(* Logix 5000 project; controller test vendor 1 type 14 code 151 rev 32.13; software revision 32.02 *)

TASK P200ms_p10 (periodic, rate 200 ms, priority 10, watchdog 300 ms) : GUI, ValveProfile
TASK P_Sample_p5 (periodic, rate 10 ms, priority 5, watchdog 2000 ms) : measArray, ISR_ValveCtrl   // Get raw analog input and control of the breathing - MUST HAVE HIGHEST priority of all peridoc tasks
TASK P_Sample_p8 (periodic, rate 10 ms, priority 8, watchdog 500 ms) : Setup, calcBreath, initVent, BreathDetect, measCalc, MainFlow

MODULES
   Local : vendor 1 type 14 code 151 (Compact 0, rev 32.13)
      Counters : Embedded (Compact 3, rev 1.1, Output RPI 20 ms)
      Discrete_IO : Embedded (Compact 1, rev 3.1, Output RPI 20 ms)
      Analog_IO : Embedded (Compact 2, rev 1.1, Output RPI 2 ms)
END_MODULES

ADD_ON_INSTRUCTION AOI_ARRAYSHIFT   (* revision 1.0, vendor RA - Brian Askjaer *)
VAR_IN_OUT
   Inp_Array : REAL[1000,2]; {required}
   _Array : REAL[1000,2]; {required}
END_VAR

ROUTINE Logic   (* ladder *)
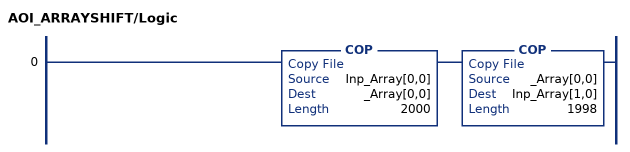
   0: COP(Inp_Array[0,0],_Array[0,0],2000)COP(_Array[0,0],Inp_Array[1,0],1998);
END_ROUTINE
END_ADD_ON_INSTRUCTION

ADD_ON_INSTRUCTION AOI_Ceil   (* revision 1.1 *)
VAR_INPUT
   In_X : REAL; {required}
END_VAR
VAR_IN_OUT
   Out_Ret : REAL; {required}
END_VAR
VAR
   _trunc : REAL; {access None}
   _aoiTrunc : AOI_Trunc; {access None}
   _n : DINT; {access None}
END_VAR

ROUTINE Logic   (* structured text *)
   AOI_Trunc( _aoiTrunc, In_X, _trunc );
   _n := _trunc;
   if _n < In_X then
   	_n := _n + 1;
   end_if;
   Out_Ret := _n;
   
END_ROUTINE
END_ADD_ON_INSTRUCTION

ADD_ON_INSTRUCTION AOI_FillArray_Real2D   (* revision 1.0, vendor RA - Brian Askjaer *)
VAR_IN_OUT
   Array : REAL[1000,2]; {required}
END_VAR
VAR_INPUT
   Source : DINT; {required}
   Len : DINT; {required}
END_VAR

ROUTINE Logic   (* ladder *)
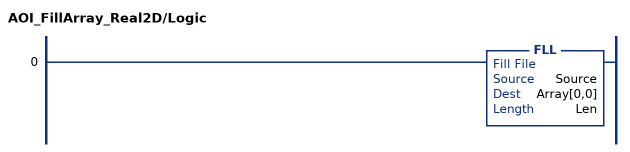
   0: FLL(Source,Array[0,0],Len);
END_ROUTINE
END_ADD_ON_INSTRUCTION

ADD_ON_INSTRUCTION AOI_FillArrayInt   (* revision 1.0, vendor RA - Brian Askjaer *)
VAR_IN_OUT
   Array : INT[1000]; {required}
END_VAR
VAR_INPUT
   Source : DINT; {required}
   Len : DINT; {required}
END_VAR

ROUTINE Logic   (* ladder *)
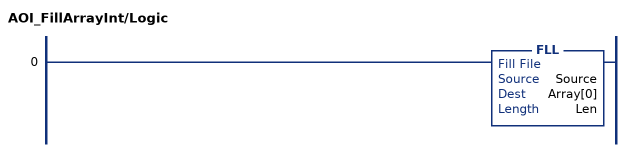
   0: FLL(Source,Array[0],Len);
END_ROUTINE
END_ADD_ON_INSTRUCTION

ADD_ON_INSTRUCTION AOI_FillArrayReal   (* revision 1.0, vendor RA - Brian Askjaer *)
VAR_IN_OUT
   Array : REAL[650]; {required}
END_VAR
VAR_INPUT
   Source : DINT; {required}
   Len : DINT; {required}
END_VAR

ROUTINE Logic   (* ladder *)
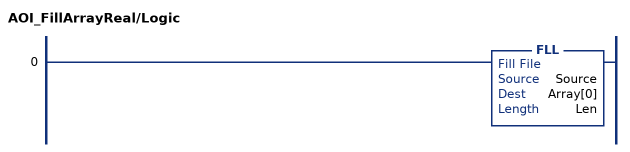
   0: FLL(Source,Array[0],Len);
END_ROUTINE
END_ADD_ON_INSTRUCTION

ADD_ON_INSTRUCTION AOI_FillArrayReal50   (* revision 1.0, vendor RA - Brian Askjaer *)
VAR_IN_OUT
   Array : REAL[50]; {required}
END_VAR
VAR_INPUT
   Source : DINT; {required}
   Len : DINT; {required}
END_VAR

ROUTINE Logic   (* ladder *)
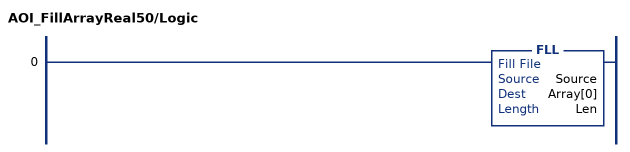
   0: FLL(Source,Array[0],Len);
END_ROUTINE
END_ADD_ON_INSTRUCTION

ADD_ON_INSTRUCTION AOI_FilterSignal   (* revision 1.1, ExecutePrescan *)
VAR_INPUT
   In_rRawSignal : REAL; {required}
   In_bInitialize : BOOL; {visible}
   Par_eType : DINT; {visible}   // 0: MEDIAN; 1: MEAN
   Par_nWindowLeft : DINT; {visible}
   Par_nWindowsRight : DINT; {visible}
   Par_bUseWeights : BOOL; {visible}   // Used for mean filtering
END_VAR
VAR_IN_OUT
   Par_rWeights : REAL[1]; {required}   // Used for mean filtering
END_VAR
VAR_OUTPUT
   Out_Buffering : BOOL; {visible}
   Out_rFilteredSignalDelayed : REAL; {access Read Only, visible}
   ER : BOOL; {access Read Only, visible}
   Err : DINT; {visible}
END_VAR
VAR
   _n1 : DINT; {access None}
   _n0 : DINT; {access None}
   _nN : DINT; {access None}
   _nM : DINT; {access None}
   _rWs : REAL[31]; {access None}
   _bW : BOOL; {access None}
   _idx : DINT; {access None}
   _bFirstScan : BOOL; {access None}
   _nTmp : DINT; {access None}
   _rRawBuf : REAL[31]; {access None}
   _eType : DINT; {access None}
   _srt : CONTROL; {access None}
   _nBufferUsage : DINT; {access None}
   _rBufSorted : REAL[31]; {access None}
   _i : DINT; {access None}
   _rSum : REAL; {access None}
   _w : REAL; {access None}
   _nOff : DINT; {access None}
   _n2 : DINT; {access None}
   _bOdd : BOOL; {access None}
   _rSumW : REAL; {access None}
END_VAR

ROUTINE Logic   (* structured text *)
   if ER and not ( _bFirstScan or In_bInitialize ) then
   	tnd();
   end_if;
   
   // Initialization
   if In_bInitialize or _bFirstScan then
   	ER  := 0;
   	Err := 0;
   	_idx := 0;
   	_nBufferUsage := 0;
   
   	// Validate parameters
   	_nTmp := Par_nWindowLeft + Par_nWindowsRight + 1;
   	if Par_nWindowLeft   < 0 then Err := 1; end_if;
   	if Par_nWindowsRight < 0 then Err := 2; end_if;
   	if _nTmp > _nM  then Err := 3; end_if;
   	if Par_eType <> 0 and Par_eType <> 1 then Err := 4; end_if;
   	if Err <> 0 then
   		ER := 1;
   		tnd();
   	end_if;
   
   	// Store parameters ( make filter behaviour independent from outside
   	//   parameters' changes ).
   	_bW := Par_bUseWeights;
   	_n0 := Par_nWindowLeft;
   	_n1 := Par_nWindowsRight;
   	_nN := _nTmp;
   	_n2 := _nN / 2;
   	_bOdd := ( _nN mod 2 ) = 1; // neighbourhood window composed of a odd number of points
   	_eType := Par_eType;
   	cop( Par_rWeights[0], _rWs[0], _nN );
   	_srt.POS := 0;
   	_srt.LEN := _nN;
   	_w := 1.0;
   	_rSumW := _nN;
   	if _bW then
   		_rSumW := 0.0;
   		for _i := 0 to _nN - 1 do
   			_rSumW := _rSumW + _rWs[_i];
   		end_for;
   	end_if;
   
   end_if;
   _bFirstScan := 0;
   In_bInitialize := 0;
   
   // While buffering data the filter isn't applied
   _rRawBuf[ _idx ] := In_rRawSignal;
   if _nBufferUsage < _nN then _nBufferUsage := _nBufferUsage + 1; end_if;
   Out_Buffering := _nBufferUsage <> _nN;
   
   if not Out_Buffering then
   
   	case _eType of
   
   		0: // MEDIAN
   		// Very simple implementation but not very efficient.
   		//   It's ok here because a single filtered value is
   		//   calculated at every scan of the plc.
   		// I'm using firmware instruction SRT to
   		//   sort the buffer array, because it's faster
   		//   than anything that could be implemented in
   		//   structure text. In case SRT isn't available in
   		//   other PLCs, a sorting algorithm could be implemented.
   		//   For example, in file sort/sort.c of the Gnu Scientific
   		//     Library (ftp://ftp.gnu.org/gnu/gsl/) there is an
   		//     implementation of the heap sort algorithm.
   		// TODO: replace the SRT instruction with such GLS
   		//       implementation so that this code can be reused
   		//       in any PLC.
   		cop( _rRawBuf[0], _rBufSorted[0], _nN );
   		SRT( _rBufSorted, 0, _srt );
   		if _bOdd then
   			Out_rFilteredSignalDelayed := _rBufSorted[_n2];
   		else
   			Out_rFilteredSignalDelayed := 0.5 * ( _rBufSorted[_n2-1] + _rBufSorted[_n2] );
   		end_if;
   
   		1: // MEAN
   		// Note: instruction MAVE could be used here, but I find
   		//       the following code clearer. Moreover the code
   		//       can be used in any PLC which doesn't include the
   		//       MAVE instruction.
   		_rSum := 0.0;
   		for _i := 0 to _nN - 1 do
   			if _bW then _w := _rWs[_i]; end_if;
   			_rSum := _rSum + _w * _rRawBuf[ ( _idx + 1 + _i ) mod _nN ];
   		end_for;
   		Out_rFilteredSignalDelayed := _rSum / _rSumW;
   
   	end_case;
   
   end_if;
   
   _idx := ( _idx + 1 ) mod _nN;
   
END_ROUTINE

ROUTINE Prescan   (* structured text *)
   // Calulate _nN = minimum between size( Par_rWeights ), size(_rWs), size(_rBuf) and size(_rBufSorted)
   size( _rWs, 0, _nM );
   size( _rRawBuf, 0, _nTmp );
   if _nTmp < _nM then _nM := _nTmp; end_if;
   size( _rBufSorted, 0, _nTmp );
   if _nTmp < _nM then _nM := _nTmp; end_if;
   size( Par_rWeights, 0, _nTmp );
   if _nTmp < _nM then _nM := _nTmp; end_if;
   
   // Used for initialization
   _bFirstScan := 1;
   
   // Data must be buffered at the beginning
   Out_Buffering := 1;
   
END_ROUTINE
END_ADD_ON_INSTRUCTION

ADD_ON_INSTRUCTION AOI_Floor   (* revision 1.1 *)
VAR_INPUT
   In_X : REAL; {required}
END_VAR
VAR_IN_OUT
   Out_Ret : REAL; {required}
END_VAR
VAR
   _n : DINT; {access None}
   _ret : REAL; {access None}
END_VAR

ROUTINE Logic   (* structured text *)
   _n := In_X;
   if In_X < _n then
   	_ret := _n - 1;
   else
   	_ret := _n;
   end_if;
   Out_Ret := _ret;
   
END_ROUTINE
END_ADD_ON_INSTRUCTION

ADD_ON_INSTRUCTION AOI_Max   (* revision 1.0, ExecutePrescan *)
VAR_IN_OUT
   In_Array : REAL[1000,2]; {required}
END_VAR
VAR_INPUT
   In_MainIndex : DINT; {required}
   In_N0 : INT; {required}
   In_N1 : INT; {required}
END_VAR
VAR_OUTPUT
   Out_Max : REAL; {visible}
   Err : DINT; {visible}
   ER : BOOL; {visible}
END_VAR
VAR_INPUT
   _i : DINT;
END_VAR
VAR
   _maxDim0 : DINT; {access None}
   _maxDim1 : DINT;
   _max : REAL; {access None}
   _tmp : REAL; {access None}
END_VAR

ROUTINE Logic   (* structured text *)
   ER  := 0;
   Err := 0;
   
   // Some checks
   if In_MainIndex < 0 or _maxDim1 <= In_MainIndex then Err := 1; end_if;
   if In_N0 < 0        or _maxDim0 <= In_N0        then Err := 2; end_if;
   if In_N1 < 0        or _maxDim0 <= In_N1        then Err := 3; end_if;
   if In_N0 > In_N1                                then Err := 4; end_if;
   if Err <> 0 then
   	ER := 1;
   	tnd();
   end_if;
   
   // Find maximum
   _max := In_Array[ In_N0, In_MainIndex ];
   for _i := In_N0 + 1 to In_N1 do
   	_tmp := In_Array[ _i, In_MainIndex ];
   	if _max < _tmp then _max := _tmp; end_if;
   end_for;
   Out_Max := _max;
   
END_ROUTINE

ROUTINE Prescan   (* structured text *)
   size( In_Array, 0, _maxDim0 ); // Dimension 0 is the most right index
   size( In_Array, 1, _maxDim1 );
   
END_ROUTINE
END_ADD_ON_INSTRUCTION

ADD_ON_INSTRUCTION AOI_Mean2D   (* revision 1.0, ExecutePrescan *)
VAR_IN_OUT
   In_Array : REAL[1000,2]; {required}
END_VAR
VAR_INPUT
   In_MainIndex : DINT; {required}
   In_N0 : INT; {required}
   In_N1 : INT; {required}
END_VAR
VAR_OUTPUT
   Out_Mean : REAL; {visible}
   Err : DINT; {visible}
   ER : BOOL; {visible}
END_VAR
VAR_INPUT
   _i : DINT;
END_VAR
VAR
   _maxDim0 : DINT; {access None}
   _maxDim1 : DINT;
   _sum : REAL; {access None}
END_VAR

ROUTINE Logic   (* structured text *)
   ER  := 0;
   Err := 0;
   
   // Some checks
   if In_MainIndex < 0 or _maxDim1 <= In_MainIndex then Err := 1; end_if;
   if In_N0 < 0        or _maxDim0 <= In_N0        then Err := 2; end_if;
   if In_N1 < 0        or _maxDim0 <= In_N1        then Err := 3; end_if;
   if In_N0 > In_N1                                then Err := 4; end_if;
   if Err <> 0 then
   	ER := 1;
   	tnd();
   end_if;
   
   // Find mean
   _sum := 0.0;
   for _i := In_N0 to In_N1 do
   	_sum := _sum + In_Array[ _i, In_MainIndex ];
   end_for;
   Out_Mean := _sum / ( In_N1 - In_N0 + 1 );
   
END_ROUTINE

ROUTINE Prescan   (* structured text *)
   size( In_Array, 0, _maxDim0 ); // Dimension 0 is the most right index
   size( In_Array, 1, _maxDim1 );
   
END_ROUTINE
END_ADD_ON_INSTRUCTION

ADD_ON_INSTRUCTION AOI_Mean50   (* revision 1.0, ExecutePrescan *)
VAR_IN_OUT
   In_Array : REAL[50]; {required}
END_VAR
VAR_INPUT
   In_N0 : INT; {required}
   In_N1 : INT; {required}
END_VAR
VAR_OUTPUT
   Out_Mean : REAL; {visible}
   Err : DINT; {visible}
   ER : BOOL; {visible}
END_VAR
VAR_INPUT
   _i : DINT;
END_VAR
VAR
   _maxDim0 : DINT; {access None}
   _maxDim1 : DINT;
   _sum : REAL; {access None}
END_VAR

ROUTINE Logic   (* structured text *)
   ER  := 0;
   Err := 0;
   
   // Some checks
   if In_N0 < 0        or _maxDim0 <= In_N0        then Err := 2; end_if;
   if In_N1 < 0        or _maxDim0 <= In_N1        then Err := 3; end_if;
   if In_N0 > In_N1                                then Err := 4; end_if;
   if Err <> 0 then
   	ER := 1;
   	tnd();
   end_if;
   
   // Find mean
   _sum := 0.0;
   for _i := In_N0 to In_N1 do
   	_sum := _sum + In_Array[ _i];
   end_for;
   Out_Mean := _sum / ( In_N1 - In_N0 + 1 );
   
END_ROUTINE

ROUTINE Prescan   (* structured text *)
   size( In_Array, 0, _maxDim0 ); // Dimension 0 is the most right index
   
END_ROUTINE
END_ADD_ON_INSTRUCTION

ADD_ON_INSTRUCTION AOI_Round   (* revision 1.0 *)
VAR_INPUT
   In_X : REAL; {required}
END_VAR
VAR_IN_OUT
   Out_Ret : REAL; {required}
END_VAR
VAR
   _n : DINT; {access None}
END_VAR

ROUTINE Logic   (* structured text *)
   _n := In_X;
   Out_Ret := _n;
   
END_ROUTINE
END_ADD_ON_INSTRUCTION

ADD_ON_INSTRUCTION AOI_Trunc   (* revision 1.0 *)
VAR_INPUT
   In_X : REAL; {required}
END_VAR
VAR_IN_OUT
   Out_Ret : REAL; {required}
END_VAR

ROUTINE Logic   (* structured text *)
   // TODO: Logix has a truc function but other PLCs may not.
   //       Replace the native function in Logix with an
   //       implementation which will work with other PLC.
   //       Note that AOI_Trunc and AOI_Ceil (which depends
   //       on AOI_Trunc ) may not be needed in the project.
   
   Out_Ret := trunc( In_X );
   
END_ROUTINE
END_ADD_ON_INSTRUCTION

VAR_GLOBAL   (* controller tags *)
   _CopDes1 : DINT;
   _CopDes4 : DINT;
   _CopDes5 : DINT;
   _CopDes6 : DINT;
   _CopDes8 : DINT;
   _CopLength : DINT;
   _CopLength1 : DINT;
   _CopLength3 : DINT;
   _CopLength4 : DINT;
   _CopLength5 : DINT;
   _CopLength6 : DINT;
   _CopLength7 : DINT := 2060;
   _CopLength8 : DINT;
   _CopSource : DINT;
   _CopSource1 : DINT;
   _CopSource3 : DINT;
   _CopSource4 : DINT;
   _CopSource5 : DINT;
   _CopSource6 : DINT;
   _CopSource7 : DINT := -30;
   _CopSource8 : DINT;
   _edbAoiFilterFlowAir : AOI_FilterSignal := (In_rRawSignal := 982.0, Par_nWindowLeft := 5, Par_nWindowsRight := 5, Out_rFilteredSignalDelayed := 982.0);
   _edbAoiFilterFlowO2 : AOI_FilterSignal := (In_rRawSignal := 983.0, Par_nWindowLeft := 5, Par_nWindowsRight := 5, Out_rFilteredSignalDelayed := 984.0);
   _edbAoiFilterPress : AOI_FilterSignal := (In_rRawSignal := 3963.0, Par_nWindowLeft := 5, Par_nWindowsRight := 5, Out_rFilteredSignalDelayed := 3951.0);
   _edbCanStore : BOOL := 1;
   _edbFlowArrFiltered : REAL[1000,2] := ([5,0] := 982.0, [6,0] := 982.0, [7,0] := 982.0, [8,0] := 982.0, [9,0] := 982.0, [10,0] := 982.0, [11,0] := 982.0, [12,0] := 982.0, [13,0] := 982.0, [14,0] := 982.0, [15,0] := 983.0, [16,0] := 983.0, [17,0] := 982.0, [18,0] := 982.0, [19,0] := 982.0, [20,0] := 982.0, [21,0] := 982.0, [22,0] := 982.0, [23,0] := 982.0, [24,0] := 982.0, [25,0] := 982.0, [26,0] := 982.0, [27,0] := 982.0, [28,0] := 982.0, [29,0] := 982.0, [30,0] := 982.0, [31,0] := 982.0, [32,0] := 982.0, [33,0] := 982.0, [34,0] := 982.0, [35,0] := 982.0, [36,0] := 982.0, [37,0] := 982.0, [38,0] := 982.0, [39,0] := 982.0, [40,0] := 982.0, [41,0] := 982.0, [42,0] := 982.0, [43,0] := 983.0, [44,0] := 983.0, [45,0] := 983.0, [46,0] := 983.0, [47,0] := 983.0, [48,0] := 983.0, [49,0] := 982.0, [50,0] := 982.0, [51,0] := 982.0, [52,0] := 982.0, [53,0] := 982.0, [54,0] := 982.0, [55,0] := 982.0, [56,0] := 982.0, [57,0] := 982.0, [58,0] := 982.0, [59,0] := 982.0, [60,0] := 982.0, [61,0] := 982.0, [62,0] := 982.0, [63,0] := 982.0, [64,0] := 982.0,
        [65,0] := 982.0, [66,0] := 982.0, [67,0] := 982.0, [68,0] := 982.0, [69,0] := 982.0, [70,0] := 982.0, [71,0] := 982.0, [72,0] := 982.0, [73,0] := 982.0, [74,0] := 982.0, [75,0] := 982.0, [76,0] := 982.0, [77,0] := 983.0, [78,0] := 983.0, [79,0] := 982.0, [80,0] := 982.0, [81,0] := 982.0, [82,0] := 982.0, [83,0] := 982.0, [84,0] := 982.0, [85,0] := 982.0, [86,0] := 982.0, [87,0] := 982.0, [88,0] := 982.0, [89,0] := 982.0, [90,0] := 982.0, [91,0] := 982.0, [92,0] := 982.0, [93,0] := 982.0, [94,0] := 982.0, [95,0] := 982.0, [96,0] := 982.0, [97,0] := 982.0, [98,0] := 982.0, [99,0] := 982.0, [100,0] := 982.0, [101,0] := 982.0, [102,0] := 982.0, [103,0] := 982.0, [104,0] := 982.0, [105,0] := 982.0, [106,0] := 982.0, [107,0] := 982.0, [108,0] := 982.0, [109,0] := 982.0, [110,0] := 982.0, [111,0] := 982.0, [112,0] := 982.0, [113,0] := 983.0, [114,0] := 983.0, [115,0] := 983.0, [116,0] := 983.0, [117,0] := 983.0, [118,0] := 982.0, [119,0] := 982.0, [120,0] := 982.0, [121,0] := 982.0, [122,0] := 982.0, [123,0] := 982.0, [124,0] := 982.0,
        [125,0] := 982.0, [126,0] := 982.0, [127,0] := 982.0, [128,0] := 982.0, [129,0] := 982.0, [130,0] := 982.0, [131,0] := 982.0, [132,0] := 982.0, [133,0] := 982.0, [134,0] := 982.0, [135,0] := 982.0, [136,0] := 982.0, [137,0] := 982.0, [138,0] := 982.0, [139,0] := 982.0, [140,0] := 982.0, [141,0] := 982.0, [142,0] := 982.0, [143,0] := 982.0, [144,0] := 983.0, [145,0] := 983.0, [146,0] := 983.0, [147,0] := 983.0, [148,0] := 983.0, [149,0] := 983.0, [150,0] := 982.0, [151,0] := 982.0, [152,0] := 982.0, [153,0] := 982.0, [154,0] := 982.0, [155,0] := 982.0, [156,0] := 982.0, [157,0] := 982.0, [158,0] := 982.0, [159,0] := 982.0, [160,0] := 982.0, [161,0] := 982.0, [162,0] := 982.0, [163,0] := 982.0, [164,0] := 982.0, [165,0] := 982.0, [166,0] := 982.0, [167,0] := 982.0, [168,0] := 982.0, [169,0] := 982.0, [170,0] := 982.0, [171,0] := 982.0, [172,0] := 982.0, [173,0] := 982.0, [174,0] := 982.0, [175,0] := 982.0, [176,0] := 983.0, [177,0] := 983.0, [178,0] := 983.0, [179,0] := 983.0, [180,0] := 982.0, [181,0] := 982.0, [182,0] := 982.0, [183,0] := 982.0, [184,0] := 982.0,
        [185,0] := 982.0, [186,0] := 982.0, [187,0] := 982.0, [188,0] := 982.0, [189,0] := 982.0, [190,0] := 982.0, [191,0] := 982.0, [192,0] := 982.0, [193,0] := 982.0, [194,0] := 982.0, [195,0] := 982.0, [196,0] := 982.0, [197,0] := 982.0, [198,0] := 982.0, [199,0] := 982.0, [200,0] := 982.0, [201,0] := 982.0, [202,0] := 982.0, [203,0] := 982.0, [204,0] := 982.0, [205,0] := 982.0, [206,0] := 982.0, [207,0] := 982.0, [208,0] := 982.0, [209,0] := 982.0, [210,0] := 982.0, [211,0] := 982.0, [212,0] := 982.0, [213,0] := 982.0, [214,0] := 982.0, [215,0] := 982.0, [216,0] := 982.0, [217,0] := 982.0, [218,0] := 982.0, [219,0] := 982.0, [220,0] := 982.0, [221,0] := 982.0, [222,0] := 982.0, [223,0] := 982.0, [224,0] := 982.0, [225,0] := 982.0, [226,0] := 982.0, [227,0] := 982.0, [228,0] := 982.0, [229,0] := 982.0, [230,0] := 982.0, [231,0] := 982.0, [232,0] := 982.0, [233,0] := 982.0, [234,0] := 982.0, [235,0] := 982.0, [236,0] := 982.0, [237,0] := 982.0, [238,0] := 982.0, [239,0] := 982.0, [240,0] := 982.0, [241,0] := 982.0, [242,0] := 982.0, [243,0] := 982.0, [244,0] := 982.0,
        [245,0] := 982.0, [246,0] := 982.0, [247,0] := 982.0, [248,0] := 982.0, [249,0] := 982.0, [250,0] := 982.0, [251,0] := 982.0, [252,0] := 982.0, [253,0] := 982.0, [254,0] := 982.0, [255,0] := 982.0, [256,0] := 982.0, [257,0] := 982.0, [258,0] := 982.0, [259,0] := 982.0, [260,0] := 982.0, [261,0] := 982.0, [262,0] := 982.0, [263,0] := 982.0, [264,0] := 982.0, [265,0] := 982.0, [266,0] := 982.0, [267,0] := 982.0, [268,0] := 982.0, [269,0] := 982.0, [270,0] := 982.0, [271,0] := 983.0, [272,0] := 983.0, [273,0] := 983.0, [274,0] := 983.0, [275,0] := 982.0, [276,0] := 982.0, [277,0] := 982.0, [278,0] := 982.0, [279,0] := 982.0, [280,0] := 982.0, [281,0] := 982.0, [282,0] := 982.0, [283,0] := 982.0, [284,0] := 982.0, [285,0] := 982.0, [286,0] := 982.0, [287,0] := 982.0, [288,0] := 982.0, [289,0] := 982.0, [290,0] := 982.0, [291,0] := 982.0, [292,0] := 982.0, [293,0] := 982.0, [294,0] := 982.0, [295,0] := 982.0, [296,0] := 982.0, [297,0] := 982.0, [298,0] := 982.0, [299,0] := 982.0, [300,0] := 982.0, [301,0] := 982.0, [302,0] := 982.0, [303,0] := 982.0, [304,0] := 982.0,
        [305,0] := 982.0, [306,0] := 982.0, [307,0] := 982.0, [308,0] := 982.0, [309,0] := 982.0, [310,0] := 982.0, [311,0] := 982.0, [312,0] := 982.0, [313,0] := 982.0, [314,0] := 982.0, [315,0] := 982.0, [316,0] := 982.0, [317,0] := 982.0, [318,0] := 982.0, [319,0] := 982.0, [320,0] := 982.0, [321,0] := 982.0, [322,0] := 982.0, [323,0] := 982.0, [324,0] := 982.0, [325,0] := 982.0, [326,0] := 982.0, [327,0] := 982.0, [328,0] := 982.0, [329,0] := 982.0, [330,0] := 982.0, [331,0] := 982.0, [332,0] := 983.0, [333,0] := 983.0, [334,0] := 983.0, [335,0] := 983.0, [336,0] := 983.0, [337,0] := 983.0, [338,0] := 983.0, [339,0] := 983.0, [340,0] := 982.0, [341,0] := 982.0, [342,0] := 982.0, [343,0] := 982.0, [344,0] := 982.0, [345,0] := 982.0, [346,0] := 982.0, [347,0] := 982.0, [348,0] := 982.0, [349,0] := 982.0, [350,0] := 982.0, [351,0] := 982.0, [352,0] := 982.0, [353,0] := 982.0, [354,0] := 982.0, [355,0] := 982.0, [356,0] := 982.0, [357,0] := 982.0, [358,0] := 982.0, [359,0] := 982.0, [360,0] := 982.0, [361,0] := 982.0, [362,0] := 982.0, [363,0] := 982.0, [364,0] := 982.0,
        [365,0] := 982.0, [366,0] := 982.0, [367,0] := 982.0, [368,0] := 982.0, [369,0] := 982.0, [370,0] := 982.0, [371,0] := 982.0, [372,0] := 982.0, [373,0] := 982.0, [374,0] := 982.0, [375,0] := 982.0, [376,0] := 982.0, [377,0] := 982.0, [378,0] := 982.0, [379,0] := 982.0, [380,0] := 982.0, [381,0] := 982.0, [382,0] := 982.0, [383,0] := 982.0, [384,0] := 982.0, [385,0] := 982.0, [386,0] := 982.0, [387,0] := 982.0, [388,0] := 982.0, [389,0] := 982.0, [390,0] := 982.0, [391,0] := 982.0, [392,0] := 982.0, [393,0] := 982.0, [394,0] := 982.0, [395,0] := 982.0, [396,0] := 982.0, [397,0] := 982.0, [398,0] := 982.0, [399,0] := 982.0, [400,0] := 982.0, [401,0] := 982.0, [402,0] := 982.0, [403,0] := 982.0, [404,0] := 982.0, [405,0] := 982.0, [406,0] := 982.0, [407,0] := 982.0, [408,0] := 982.0, [409,0] := 982.0, [410,0] := 982.0, [411,0] := 982.0, [412,0] := 982.0, [413,0] := 982.0, [414,0] := 982.0, [415,0] := 982.0, [416,0] := 982.0, [417,0] := 982.0, [418,0] := 982.0, [419,0] := 982.0, [420,0] := 982.0, [421,0] := 982.0, [422,0] := 982.0, [423,0] := 982.0, [424,0] := 982.0,
        [425,0] := 982.0, [426,0] := 983.0, [427,0] := 983.0, [428,0] := 983.0, [429,0] := 983.0, [430,0] := 983.0, [431,0] := 982.0, [432,0] := 982.0, [433,0] := 982.0, [434,0] := 982.0, [435,0] := 982.0, [436,0] := 982.0, [437,0] := 982.0, [438,0] := 982.0, [439,0] := 982.0, [440,0] := 982.0, [441,0] := 982.0, [442,0] := 982.0, [443,0] := 982.0, [444,0] := 982.0, [445,0] := 982.0, [446,0] := 982.0, [447,0] := 982.0, [448,0] := 982.0, [449,0] := 982.0, [450,0] := 982.0, [451,0] := 982.0, [452,0] := 982.0, [453,0] := 982.0, [454,0] := 982.0, [455,0] := 982.0, [456,0] := 982.0, [457,0] := 982.0, [458,0] := 982.0, [459,0] := 982.0, [460,0] := 982.0, [461,0] := 982.0, [462,0] := 982.0, [463,0] := 982.0, [464,0] := 982.0, [465,0] := 983.0, [466,0] := 983.0, [467,0] := 983.0, [468,0] := 983.0, [469,0] := 982.0, [470,0] := 982.0, [471,0] := 982.0, [472,0] := 982.0, [473,0] := 982.0, [474,0] := 982.0, [475,0] := 982.0, [476,0] := 982.0, [477,0] := 982.0, [478,0] := 982.0, [479,0] := 982.0, [480,0] := 982.0, [481,0] := 982.0, [482,0] := 982.0, [483,0] := 982.0, [484,0] := 982.0,
        [485,0] := 982.0, [486,0] := 982.0, [487,0] := 982.0, [488,0] := 982.0, [489,0] := 982.0, [490,0] := 982.0, [491,0] := 983.0, [492,0] := 983.0, [493,0] := 982.0, [494,0] := 982.0, [495,0] := 982.0, [496,0] := 982.0, [497,0] := 983.0, [498,0] := 983.0, [499,0] := 983.0, [500,0] := 982.0, [501,0] := 982.0, [502,0] := 982.0, [503,0] := 982.0, [504,0] := 982.0, [505,0] := 982.0, [506,0] := 982.0, [507,0] := 982.0, [508,0] := 982.0, [509,0] := 982.0, [510,0] := 982.0, [511,0] := 982.0, [512,0] := 982.0, [513,0] := 982.0, [514,0] := 982.0, [515,0] := 982.0, [516,0] := 982.0, [517,0] := 982.0, [518,0] := 982.0, [519,0] := 982.0, [520,0] := 982.0, [521,0] := 982.0, [522,0] := 982.0, [523,0] := 982.0, [524,0] := 982.0, [525,0] := 982.0, [526,0] := 982.0, [527,0] := 982.0, [528,0] := 982.0, [529,0] := 982.0, [530,0] := 983.0, [531,0] := 983.0, [532,0] := 982.0, [533,0] := 982.0, [534,0] := 982.0, [535,0] := 982.0, [536,0] := 982.0, [537,0] := 982.0, [538,0] := 982.0, [539,0] := 982.0, [540,0] := 982.0, [541,0] := 982.0, [542,0] := 982.0, [543,0] := 982.0, [544,0] := 982.0,
        [545,0] := 982.0, [546,0] := 982.0, [547,0] := 982.0, [548,0] := 982.0, [549,0] := 982.0, [550,0] := 982.0, [551,0] := 982.0, [552,0] := 982.0, [553,0] := 982.0, [554,0] := 982.0, [555,0] := 982.0, [556,0] := 982.0, [557,0] := 982.0, [558,0] := 982.0, [559,0] := 982.0, [560,0] := 982.0, [561,0] := 982.0, [562,0] := 982.0, [563,0] := 982.0, [564,0] := 982.0, [565,0] := 983.0, [566,0] := 983.0, [567,0] := 983.0, [568,0] := 983.0, [569,0] := 983.0, [570,0] := 983.0, [571,0] := 983.0, [572,0] := 983.0, [573,0] := 982.0, [574,0] := 982.0, [575,0] := 982.0, [576,0] := 982.0, [577,0] := 982.0, [578,0] := 982.0, [579,0] := 982.0, [580,0] := 982.0, [581,0] := 982.0, [582,0] := 982.0, [583,0] := 982.0, [584,0] := 982.0, [585,0] := 982.0, [586,0] := 982.0, [587,0] := 982.0, [588,0] := 982.0, [589,0] := 982.0, [590,0] := 982.0, [591,0] := 982.0, [592,0] := 982.0, [593,0] := 982.0, [594,0] := 982.0, [595,0] := 982.0, [596,0] := 982.0, [597,0] := 982.0, [598,0] := 982.0, [599,0] := 982.0, [600,0] := 982.0, [601,0] := 982.0, [602,0] := 982.0, [603,0] := 982.0, [604,0] := 982.0,
        [605,0] := 982.0, [606,0] := 982.0, [607,0] := 982.0, [608,0] := 982.0, [609,0] := 982.0, [610,0] := 982.0, [611,0] := 982.0, [612,0] := 982.0, [613,0] := 982.0, [614,0] := 982.0, [615,0] := 982.0, [616,0] := 982.0, [617,0] := 982.0, [618,0] := 982.0, [619,0] := 982.0, [620,0] := 982.0, [621,0] := 982.0, [622,0] := 982.0, [623,0] := 982.0, [624,0] := 982.0, [625,0] := 982.0, [626,0] := 982.0, [627,0] := 982.0, [628,0] := 982.0, [629,0] := 982.0, [630,0] := 982.0, [631,0] := 982.0, [632,0] := 982.0, [633,0] := 982.0, [634,0] := 982.0, [635,0] := 982.0, [636,0] := 982.0, [637,0] := 982.0, [638,0] := 982.0, [639,0] := 982.0, [640,0] := 982.0, [641,0] := 982.0, [642,0] := 982.0, [643,0] := 982.0, [644,0] := 982.0, [645,0] := 982.0, [646,0] := 982.0, [647,0] := 982.0, [648,0] := 982.0, [649,0] := 982.0, [650,0] := 982.0, [651,0] := 982.0, [652,0] := 982.0, [653,0] := 982.0, [654,0] := 982.0, [655,0] := 983.0, [656,0] := 983.0, [657,0] := 982.0, [658,0] := 982.0, [659,0] := 982.0, [660,0] := 982.0, [661,0] := 982.0, [662,0] := 982.0, [663,0] := 982.0, [664,0] := 982.0,
        [665,0] := 982.0, [666,0] := 982.0, [667,0] := 982.0, [668,0] := 982.0, [669,0] := 982.0, [670,0] := 982.0, [671,0] := 982.0, [672,0] := 982.0, [673,0] := 982.0, [674,0] := 982.0, [675,0] := 982.0, [676,0] := 982.0, [677,0] := 982.0, [678,0] := 982.0, [679,0] := 982.0, [680,0] := 982.0, [681,0] := 982.0, [682,0] := 982.0, [683,0] := 982.0, [684,0] := 982.0, [685,0] := 982.0, [686,0] := 982.0, [687,0] := 982.0, [688,0] := 982.0, [689,0] := 982.0, [690,0] := 982.0, [691,0] := 982.0, [692,0] := 983.0, [693,0] := 983.0, [694,0] := 983.0, [695,0] := 983.0, [696,0] := 983.0, [697,0] := 983.0, [698,0] := 982.0, [699,0] := 982.0, [700,0] := 982.0, [701,0] := 982.0, [702,0] := 982.0, [703,0] := 982.0, [704,0] := 982.0, [705,0] := 982.0, [706,0] := 982.0, [707,0] := 982.0, [708,0] := 982.0, [709,0] := 982.0, [710,0] := 982.0, [711,0] := 982.0, [712,0] := 982.0, [713,0] := 982.0, [714,0] := 982.0, [715,0] := 982.0, [716,0] := 982.0, [717,0] := 982.0, [718,0] := 982.0, [719,0] := 982.0, [720,0] := 982.0, [721,0] := 982.0, [722,0] := 983.0, [723,0] := 983.0, [724,0] := 983.0,
        [725,0] := 983.0, [726,0] := 983.0, [727,0] := 983.0, [728,0] := 982.0, [729,0] := 982.0, [730,0] := 982.0, [731,0] := 982.0, [732,0] := 982.0, [733,0] := 982.0, [734,0] := 982.0, [735,0] := 982.0, [736,0] := 982.0, [737,0] := 982.0, [738,0] := 982.0, [739,0] := 982.0, [740,0] := 982.0, [741,0] := 982.0, [742,0] := 982.0, [743,0] := 982.0, [744,0] := 982.0, [745,0] := 982.0, [746,0] := 982.0, [747,0] := 982.0, [748,0] := 982.0, [749,0] := 982.0, [750,0] := 982.0, [751,0] := 982.0, [752,0] := 982.0, [753,0] := 983.0, [754,0] := 983.0, [755,0] := 983.0, [756,0] := 983.0, [757,0] := 983.0, [758,0] := 983.0, [759,0] := 982.0, [760,0] := 982.0, [761,0] := 982.0, [762,0] := 982.0, [763,0] := 982.0, [764,0] := 982.0, [765,0] := 982.0, [766,0] := 982.0, [767,0] := 982.0, [768,0] := 982.0, [769,0] := 982.0, [770,0] := 982.0, [771,0] := 982.0, [772,0] := 982.0, [773,0] := 982.0, [774,0] := 982.0, [775,0] := 982.0, [776,0] := 982.0, [777,0] := 982.0, [778,0] := 982.0, [779,0] := 982.0, [780,0] := 982.0, [781,0] := 982.0, [782,0] := 982.0, [783,0] := 982.0, [784,0] := 982.0,
        [785,0] := 983.0, [786,0] := 983.0, [787,0] := 983.0, [788,0] := 983.0, [789,0] := 982.0, [790,0] := 982.0, [791,0] := 982.0, [792,0] := 982.0, [793,0] := 982.0, [794,0] := 982.0, [795,0] := 982.0, [796,0] := 982.0, [797,0] := 982.0, [798,0] := 982.0, [799,0] := 982.0, [800,0] := 982.0, [801,0] := 982.0, [802,0] := 982.0, [803,0] := 982.0, [804,0] := 982.0, [805,0] := 982.0, [806,0] := 982.0, [807,0] := 982.0, [808,0] := 982.0, [809,0] := 982.0, [810,0] := 982.0, [811,0] := 982.0, [812,0] := 982.0, [813,0] := 982.0, [814,0] := 982.0, [815,0] := 982.0, [816,0] := 983.0, [817,0] := 983.0, [818,0] := 983.0, [819,0] := 983.0, [820,0] := 983.0, [821,0] := 982.0, [822,0] := 982.0, [823,0] := 982.0, [824,0] := 982.0, [825,0] := 982.0, [826,0] := 982.0, [827,0] := 982.0, [828,0] := 982.0, [829,0] := 982.0, [830,0] := 982.0, [831,0] := 982.0, [832,0] := 982.0, [833,0] := 982.0, [834,0] := 982.0, [835,0] := 982.0, [836,0] := 982.0, [837,0] := 982.0, [838,0] := 982.0, [839,0] := 982.0, [840,0] := 982.0, [841,0] := 982.0, [842,0] := 982.0, [843,0] := 982.0, [844,0] := 982.0,
        [845,0] := 982.0, [846,0] := 982.0, [847,0] := 983.0, [848,0] := 983.0, [849,0] := 983.0, [850,0] := 983.0, [851,0] := 983.0, [852,0] := 983.0, [853,0] := 982.0, [854,0] := 982.0, [855,0] := 982.0, [856,0] := 982.0, [857,0] := 982.0, [858,0] := 982.0, [859,0] := 982.0, [860,0] := 982.0, [861,0] := 982.0, [862,0] := 982.0, [863,0] := 982.0, [864,0] := 982.0, [865,0] := 982.0, [866,0] := 982.0, [867,0] := 982.0, [868,0] := 982.0, [869,0] := 982.0, [870,0] := 982.0, [871,0] := 982.0, [872,0] := 982.0, [873,0] := 982.0, [874,0] := 982.0, [875,0] := 982.0, [876,0] := 982.0, [877,0] := 982.0, [878,0] := 982.0, [879,0] := 982.0, [880,0] := 982.0, [881,0] := 982.0, [882,0] := 982.0, [883,0] := 982.0, [884,0] := 982.0, [885,0] := 982.0, [886,0] := 982.0, [887,0] := 982.0, [888,0] := 982.0, [889,0] := 982.0, [890,0] := 982.0, [891,0] := 982.0, [892,0] := 982.0, [893,0] := 982.0, [894,0] := 982.0, [895,0] := 982.0, [896,0] := 982.0, [897,0] := 982.0, [898,0] := 982.0, [899,0] := 982.0, [900,0] := 982.0, [901,0] := 982.0, [902,0] := 982.0, [903,0] := 982.0, [904,0] := 982.0,
        [905,0] := 982.0, [906,0] := 983.0, [907,0] := 983.0, [908,0] := 982.0, [909,0] := 982.0, [910,0] := 982.0, [911,0] := 982.0, [912,0] := 982.0, [913,0] := 982.0, [914,0] := 982.0, [915,0] := 982.0, [916,0] := 982.0, [917,0] := 982.0, [918,0] := 982.0, [919,0] := 982.0, [920,0] := 982.0, [921,0] := 982.0, [922,0] := 982.0, [923,0] := 982.0, [924,0] := 982.0, [925,0] := 982.0, [926,0] := 982.0, [927,0] := 982.0, [928,0] := 982.0, [929,0] := 982.0, [930,0] := 982.0, [931,0] := 982.0, [932,0] := 982.0, [933,0] := 982.0, [934,0] := 982.0, [935,0] := 982.0, [936,0] := 982.0, [937,0] := 982.0, [938,0] := 982.0, [939,0] := 982.0, [940,0] := 982.0, [941,0] := 982.0, [942,0] := 982.0, [943,0] := 982.0, [944,0] := 982.0, [945,0] := 982.0, [946,0] := 982.0, [947,0] := 982.0, [948,0] := 982.0, [949,0] := 982.0, [950,0] := 982.0, [951,0] := 982.0, [952,0] := 982.0, [953,0] := 982.0, [954,0] := 982.0, [955,0] := 982.0, [956,0] := 982.0, [957,0] := 983.0, [958,0] := 983.0, [959,0] := 982.0, [960,0] := 982.0, [961,0] := 982.0, [962,0] := 982.0, [963,0] := 982.0, [964,0] := 982.0,
        [965,0] := 982.0, [966,0] := 982.0, [967,0] := 982.0, [968,0] := 982.0, [969,0] := 982.0, [970,0] := 982.0, [971,0] := 982.0, [972,0] := 982.0, [973,0] := 982.0, [974,0] := 982.0, [975,0] := 982.0, [976,0] := 982.0, [977,0] := 982.0, [978,0] := 982.0, [979,0] := 983.0, [980,0] := 983.0, [981,0] := 983.0, [982,0] := 983.0, [983,0] := 983.0, [984,0] := 983.0, [985,0] := 983.0, [986,0] := 983.0, [987,0] := 982.0, [988,0] := 982.0, [989,0] := 982.0, [990,0] := 982.0, [991,0] := 982.0, [992,0] := 982.0, [993,0] := 982.0);
   _edbFlowO2Filtered : REAL[1000,2] := ([5,0] := 3948.0, [6,0] := 3948.0, [7,0] := 3948.0, [8,0] := 3948.0, [9,0] := 3948.0, [10,0] := 3948.0, [11,0] := 3948.0, [12,0] := 3948.0, [13,0] := 3948.0, [14,0] := 3950.0, [15,0] := 3950.0, [16,0] := 3950.0, [17,0] := 3951.0, [18,0] := 3951.0, [19,0] := 3951.0, [20,0] := 3951.0, [21,0] := 3951.0, [22,0] := 3951.0, [23,0] := 3951.0, [24,0] := 3951.0, [25,0] := 3951.0, [26,0] := 3951.0, [27,0] := 3951.0, [28,0] := 3951.0, [29,0] := 3948.0, [30,0] := 3948.0, [31,0] := 3948.0, [32,0] := 3948.0, [33,0] := 3948.0, [34,0] := 3957.0, [35,0] := 3957.0, [36,0] := 3957.0, [37,0] := 3957.0, [38,0] := 3948.0, [39,0] := 3948.0, [40,0] := 3945.0, [41,0] := 3945.0, [42,0] := 3945.0, [43,0] := 3945.0, [44,0] := 3954.0, [45,0] := 3954.0, [46,0] := 3954.0, [47,0] := 3954.0, [48,0] := 3954.0, [49,0] := 3954.0, [50,0] := 3954.0, [51,0] := 3954.0, [52,0] := 3954.0, [53,0] := 3954.0, [54,0] := 3954.0, [55,0] := 3954.0, [56,0] := 3954.0, [57,0] := 3954.0, [58,0] := 3944.0, [59,0] := 3944.0, [60,0] := 3944.0, [61,0] := 3944.0, [62,0] := 3954.0, [63,0] := 3954.0, [64,0] := 3954.0,
        [65,0] := 3954.0, [66,0] := 3954.0, [67,0] := 3956.0, [68,0] := 3956.0, [69,0] := 3956.0, [70,0] := 3956.0, [71,0] := 3956.0, [72,0] := 3956.0, [73,0] := 3956.0, [74,0] := 3956.0, [75,0] := 3956.0, [76,0] := 3956.0, [77,0] := 3956.0, [78,0] := 3956.0, [79,0] := 3962.0, [80,0] := 3962.0, [81,0] := 3962.0, [82,0] := 3962.0, [83,0] := 3962.0, [84,0] := 3962.0, [85,0] := 3962.0, [86,0] := 3962.0, [87,0] := 3962.0, [88,0] := 3962.0, [89,0] := 3962.0, [90,0] := 3962.0, [91,0] := 3955.0, [92,0] := 3955.0, [93,0] := 3955.0, [94,0] := 3955.0, [95,0] := 3955.0, [96,0] := 3955.0, [97,0] := 3955.0, [98,0] := 3955.0, [99,0] := 3955.0, [100,0] := 3955.0, [101,0] := 3955.0, [102,0] := 3955.0, [103,0] := 3953.0, [104,0] := 3953.0, [105,0] := 3953.0, [106,0] := 3953.0, [107,0] := 3953.0, [108,0] := 3953.0, [109,0] := 3953.0, [110,0] := 3953.0, [111,0] := 3953.0, [112,0] := 3953.0, [113,0] := 3953.0, [114,0] := 3953.0, [115,0] := 3953.0, [116,0] := 3953.0, [117,0] := 3953.0, [118,0] := 3953.0, [119,0] := 3953.0, [120,0] := 3951.0, [121,0] := 3951.0, [122,0] := 3951.0, [123,0] := 3951.0, [124,0] := 3951.0,
        [125,0] := 3951.0, [126,0] := 3951.0, [127,0] := 3951.0, [128,0] := 3953.0, [129,0] := 3953.0, [130,0] := 3953.0, [131,0] := 3953.0, [132,0] := 3953.0, [133,0] := 3953.0, [134,0] := 3953.0, [135,0] := 3954.0, [136,0] := 3954.0, [137,0] := 3954.0, [138,0] := 3954.0, [139,0] := 3949.0, [140,0] := 3949.0, [141,0] := 3949.0, [142,0] := 3949.0, [143,0] := 3949.0, [144,0] := 3949.0, [145,0] := 3949.0, [146,0] := 3949.0, [147,0] := 3949.0, [148,0] := 3949.0, [149,0] := 3949.0, [150,0] := 3949.0, [151,0] := 3949.0, [152,0] := 3951.0, [153,0] := 3951.0, [154,0] := 3951.0, [155,0] := 3951.0, [156,0] := 3951.0, [157,0] := 3954.0, [158,0] := 3954.0, [159,0] := 3951.0, [160,0] := 3951.0, [161,0] := 3951.0, [162,0] := 3951.0, [163,0] := 3951.0, [164,0] := 3954.0, [165,0] := 3954.0, [166,0] := 3954.0, [167,0] := 3954.0, [168,0] := 3944.0, [169,0] := 3944.0, [170,0] := 3944.0, [171,0] := 3944.0, [172,0] := 3944.0, [173,0] := 3944.0, [174,0] := 3956.0, [175,0] := 3956.0, [176,0] := 3948.0, [177,0] := 3948.0, [178,0] := 3948.0, [179,0] := 3948.0, [180,0] := 3952.0, [181,0] := 3952.0, [182,0] := 3952.0, [183,0] := 3952.0, [184,0] := 3952.0,
        [185,0] := 3952.0, [186,0] := 3948.0, [187,0] := 3948.0, [188,0] := 3947.0, [189,0] := 3947.0, [190,0] := 3947.0, [191,0] := 3947.0, [192,0] := 3947.0, [193,0] := 3947.0, [194,0] := 3947.0, [195,0] := 3947.0, [196,0] := 3947.0, [197,0] := 3947.0, [198,0] := 3947.0, [199,0] := 3947.0, [200,0] := 3949.0, [201,0] := 3949.0, [202,0] := 3949.0, [203,0] := 3949.0, [204,0] := 3942.0, [205,0] := 3942.0, [206,0] := 3942.0, [207,0] := 3942.0, [208,0] := 3942.0, [209,0] := 3942.0, [210,0] := 3959.0, [211,0] := 3959.0, [212,0] := 3951.0, [213,0] := 3951.0, [214,0] := 3951.0, [215,0] := 3951.0, [216,0] := 3959.0, [217,0] := 3959.0, [218,0] := 3959.0, [219,0] := 3959.0, [220,0] := 3951.0, [221,0] := 3951.0, [222,0] := 3949.0, [223,0] := 3949.0, [224,0] := 3949.0, [225,0] := 3949.0, [226,0] := 3949.0, [227,0] := 3949.0, [228,0] := 3949.0, [229,0] := 3954.0, [230,0] := 3954.0, [231,0] := 3954.0, [232,0] := 3954.0, [233,0] := 3954.0, [234,0] := 3954.0, [235,0] := 3954.0, [236,0] := 3954.0, [237,0] := 3954.0, [238,0] := 3954.0, [239,0] := 3954.0, [240,0] := 3954.0, [241,0] := 3949.0, [242,0] := 3949.0, [243,0] := 3949.0, [244,0] := 3949.0,
        [245,0] := 3960.0, [246,0] := 3960.0, [247,0] := 3960.0, [248,0] := 3960.0, [249,0] := 3960.0, [250,0] := 3960.0, [251,0] := 3953.0, [252,0] := 3953.0, [253,0] := 3954.0, [254,0] := 3954.0, [255,0] := 3954.0, [256,0] := 3954.0, [257,0] := 3954.0, [258,0] := 3954.0, [259,0] := 3954.0, [260,0] := 3954.0, [261,0] := 3954.0, [262,0] := 3954.0, [263,0] := 3954.0, [264,0] := 3954.0, [265,0] := 3953.0, [266,0] := 3953.0, [267,0] := 3953.0, [268,0] := 3953.0, [269,0] := 3953.0, [270,0] := 3952.0, [271,0] := 3952.0, [272,0] := 3952.0, [273,0] := 3952.0, [274,0] := 3952.0, [275,0] := 3952.0, [276,0] := 3952.0, [277,0] := 3947.0, [278,0] := 3947.0, [279,0] := 3947.0, [280,0] := 3947.0, [281,0] := 3947.0, [282,0] := 3955.0, [283,0] := 3955.0, [284,0] := 3955.0, [285,0] := 3955.0, [286,0] := 3945.0, [287,0] := 3945.0, [288,0] := 3945.0, [289,0] := 3945.0, [290,0] := 3945.0, [291,0] := 3945.0, [292,0] := 3954.0, [293,0] := 3954.0, [294,0] := 3953.0, [295,0] := 3953.0, [296,0] := 3953.0, [297,0] := 3953.0, [298,0] := 3954.0, [299,0] := 3954.0, [300,0] := 3954.0, [301,0] := 3954.0, [302,0] := 3954.0, [303,0] := 3954.0, [304,0] := 3953.0,
        [305,0] := 3953.0, [306,0] := 3954.0, [307,0] := 3954.0, [308,0] := 3954.0, [309,0] := 3954.0, [310,0] := 3954.0, [311,0] := 3956.0, [312,0] := 3956.0, [313,0] := 3956.0, [314,0] := 3956.0, [315,0] := 3956.0, [316,0] := 3956.0, [317,0] := 3956.0, [318,0] := 3962.0, [319,0] := 3962.0, [320,0] := 3962.0, [321,0] := 3962.0, [322,0] := 3951.0, [323,0] := 3951.0, [324,0] := 3951.0, [325,0] := 3951.0, [326,0] := 3951.0, [327,0] := 3951.0, [328,0] := 3954.0, [329,0] := 3954.0, [330,0] := 3954.0, [331,0] := 3954.0, [332,0] := 3954.0, [333,0] := 3954.0, [334,0] := 3954.0, [335,0] := 3954.0, [336,0] := 3954.0, [337,0] := 3954.0, [338,0] := 3954.0, [339,0] := 3958.0, [340,0] := 3958.0, [341,0] := 3958.0, [342,0] := 3958.0, [343,0] := 3958.0, [344,0] := 3958.0, [345,0] := 3954.0, [346,0] := 3954.0, [347,0] := 3956.0, [348,0] := 3956.0, [349,0] := 3956.0, [350,0] := 3956.0, [351,0] := 3956.0, [352,0] := 3956.0, [353,0] := 3956.0, [354,0] := 3956.0, [355,0] := 3956.0, [356,0] := 3956.0, [357,0] := 3956.0, [358,0] := 3956.0, [359,0] := 3956.0, [360,0] := 3956.0, [361,0] := 3956.0, [362,0] := 3956.0, [363,0] := 3957.0, [364,0] := 3957.0,
        [365,0] := 3957.0, [366,0] := 3957.0, [367,0] := 3957.0, [368,0] := 3957.0, [369,0] := 3957.0, [370,0] := 3957.0, [371,0] := 3957.0, [372,0] := 3957.0, [373,0] := 3957.0, [374,0] := 3957.0, [375,0] := 3957.0, [376,0] := 3957.0, [377,0] := 3957.0, [378,0] := 3957.0, [379,0] := 3957.0, [380,0] := 3957.0, [381,0] := 3949.0, [382,0] := 3949.0, [383,0] := 3948.0, [384,0] := 3948.0, [385,0] := 3948.0, [386,0] := 3948.0, [387,0] := 3942.0, [388,0] := 3942.0, [389,0] := 3942.0, [390,0] := 3942.0, [391,0] := 3946.0, [392,0] := 3946.0, [393,0] := 3948.0, [394,0] := 3948.0, [395,0] := 3946.0, [396,0] := 3946.0, [397,0] := 3946.0, [398,0] := 3946.0, [399,0] := 3946.0, [400,0] := 3950.0, [401,0] := 3950.0, [402,0] := 3950.0, [403,0] := 3950.0, [404,0] := 3949.0, [405,0] := 3949.0, [406,0] := 3949.0, [407,0] := 3949.0, [408,0] := 3949.0, [409,0] := 3949.0, [410,0] := 3950.0, [411,0] := 3950.0, [412,0] := 3957.0, [413,0] := 3957.0, [414,0] := 3957.0, [415,0] := 3957.0, [416,0] := 3957.0, [417,0] := 3957.0, [418,0] := 3957.0, [419,0] := 3957.0, [420,0] := 3957.0, [421,0] := 3957.0, [422,0] := 3957.0, [423,0] := 3957.0, [424,0] := 3945.0,
        [425,0] := 3945.0, [426,0] := 3945.0, [427,0] := 3945.0, [428,0] := 3951.0, [429,0] := 3951.0, [430,0] := 3951.0, [431,0] := 3951.0, [432,0] := 3951.0, [433,0] := 3951.0, [434,0] := 3951.0, [435,0] := 3951.0, [436,0] := 3951.0, [437,0] := 3951.0, [438,0] := 3951.0, [439,0] := 3951.0, [440,0] := 3956.0, [441,0] := 3956.0, [442,0] := 3956.0, [443,0] := 3956.0, [444,0] := 3952.0, [445,0] := 3952.0, [446,0] := 3952.0, [447,0] := 3955.0, [448,0] := 3955.0, [449,0] := 3955.0, [450,0] := 3955.0, [451,0] := 3955.0, [452,0] := 3955.0, [453,0] := 3955.0, [454,0] := 3955.0, [455,0] := 3955.0, [456,0] := 3955.0, [457,0] := 3955.0, [458,0] := 3960.0, [459,0] := 3960.0, [460,0] := 3960.0, [461,0] := 3960.0, [462,0] := 3955.0, [463,0] := 3955.0, [464,0] := 3955.0, [465,0] := 3955.0, [466,0] := 3955.0, [467,0] := 3955.0, [468,0] := 3955.0, [469,0] := 3955.0, [470,0] := 3955.0, [471,0] := 3955.0, [472,0] := 3955.0, [473,0] := 3955.0, [474,0] := 3957.0, [475,0] := 3957.0, [476,0] := 3957.0, [477,0] := 3960.0, [478,0] := 3960.0, [479,0] := 3960.0, [480,0] := 3960.0, [481,0] := 3960.0, [482,0] := 3960.0, [483,0] := 3960.0, [484,0] := 3960.0,
        [485,0] := 3960.0, [486,0] := 3960.0, [487,0] := 3963.0, [488,0] := 3963.0, [489,0] := 3959.0, [490,0] := 3959.0, [491,0] := 3959.0, [492,0] := 3959.0, [493,0] := 3959.0, [494,0] := 3957.0, [495,0] := 3957.0, [496,0] := 3957.0, [497,0] := 3957.0, [498,0] := 3957.0, [499,0] := 3951.0, [500,0] := 3951.0, [501,0] := 3946.0, [502,0] := 3946.0, [503,0] := 3946.0, [504,0] := 3946.0, [505,0] := 3946.0, [506,0] := 3946.0, [507,0] := 3946.0, [508,0] := 3946.0, [509,0] := 3946.0, [510,0] := 3937.0, [511,0] := 3937.0, [512,0] := 3935.0, [513,0] := 3935.0, [514,0] := 3952.0, [515,0] := 3952.0, [516,0] := 3952.0, [517,0] := 3947.0, [518,0] := 3947.0, [519,0] := 3947.0, [520,0] := 3947.0, [521,0] := 3947.0, [522,0] := 3947.0, [523,0] := 3952.0, [524,0] := 3952.0, [525,0] := 3949.0, [526,0] := 3949.0, [527,0] := 3949.0, [528,0] := 3949.0, [529,0] := 3949.0, [530,0] := 3949.0, [531,0] := 3949.0, [532,0] := 3949.0, [533,0] := 3949.0, [534,0] := 3949.0, [535,0] := 3949.0, [536,0] := 3949.0, [537,0] := 3949.0, [538,0] := 3949.0, [539,0] := 3949.0, [540,0] := 3949.0, [541,0] := 3949.0, [542,0] := 3959.0, [543,0] := 3959.0, [544,0] := 3959.0,
        [545,0] := 3959.0, [546,0] := 3947.0, [547,0] := 3947.0, [548,0] := 3947.0, [549,0] := 3947.0, [550,0] := 3947.0, [551,0] := 3947.0, [552,0] := 3947.0, [553,0] := 3947.0, [554,0] := 3947.0, [555,0] := 3947.0, [556,0] := 3947.0, [557,0] := 3947.0, [558,0] := 3953.0, [559,0] := 3953.0, [560,0] := 3953.0, [561,0] := 3953.0, [562,0] := 3953.0, [563,0] := 3953.0, [564,0] := 3953.0, [565,0] := 3953.0, [566,0] := 3947.0, [567,0] := 3947.0, [568,0] := 3947.0, [569,0] := 3947.0, [570,0] := 3947.0, [571,0] := 3947.0, [572,0] := 3947.0, [573,0] := 3947.0, [574,0] := 3947.0, [575,0] := 3948.0, [576,0] := 3948.0, [577,0] := 3948.0, [578,0] := 3948.0, [579,0] := 3948.0, [580,0] := 3948.0, [581,0] := 3948.0, [582,0] := 3948.0, [583,0] := 3948.0, [584,0] := 3948.0, [585,0] := 3948.0, [586,0] := 3948.0, [587,0] := 3948.0, [588,0] := 3947.0, [589,0] := 3947.0, [590,0] := 3959.0, [591,0] := 3959.0, [592,0] := 3959.0, [593,0] := 3959.0, [594,0] := 3959.0, [595,0] := 3950.0, [596,0] := 3950.0, [597,0] := 3950.0, [598,0] := 3950.0, [599,0] := 3952.0, [600,0] := 3952.0, [601,0] := 3952.0, [602,0] := 3952.0, [603,0] := 3952.0, [604,0] := 3952.0,
        [605,0] := 3951.0, [606,0] := 3951.0, [607,0] := 3951.0, [608,0] := 3951.0, [609,0] := 3951.0, [610,0] := 3951.0, [611,0] := 3951.0, [612,0] := 3951.0, [613,0] := 3951.0, [614,0] := 3951.0, [615,0] := 3951.0, [616,0] := 3951.0, [617,0] := 3951.0, [618,0] := 3951.0, [619,0] := 3954.0, [620,0] := 3954.0, [621,0] := 3954.0, [622,0] := 3954.0, [623,0] := 3956.0, [624,0] := 3956.0, [625,0] := 3956.0, [626,0] := 3956.0, [627,0] := 3956.0, [628,0] := 3956.0, [629,0] := 3954.0, [630,0] := 3954.0, [631,0] := 3943.0, [632,0] := 3943.0, [633,0] := 3943.0, [634,0] := 3943.0, [635,0] := 3943.0, [636,0] := 3943.0, [637,0] := 3943.0, [638,0] := 3943.0, [639,0] := 3943.0, [640,0] := 3945.0, [641,0] := 3945.0, [642,0] := 3945.0, [643,0] := 3947.0, [644,0] := 3947.0, [645,0] := 3947.0, [646,0] := 3947.0, [647,0] := 3947.0, [648,0] := 3947.0, [649,0] := 3947.0, [650,0] := 3947.0, [651,0] := 3947.0, [652,0] := 3950.0, [653,0] := 3950.0, [654,0] := 3950.0, [655,0] := 3950.0, [656,0] := 3950.0, [657,0] := 3950.0, [658,0] := 3950.0, [659,0] := 3955.0, [660,0] := 3955.0, [661,0] := 3955.0, [662,0] := 3955.0, [663,0] := 3955.0, [664,0] := 3959.0,
        [665,0] := 3959.0, [666,0] := 3959.0, [667,0] := 3959.0, [668,0] := 3959.0, [669,0] := 3959.0, [670,0] := 3959.0, [671,0] := 3959.0, [672,0] := 3956.0, [673,0] := 3956.0, [674,0] := 3956.0, [675,0] := 3956.0, [676,0] := 3949.0, [677,0] := 3949.0, [678,0] := 3949.0, [679,0] := 3949.0, [680,0] := 3949.0, [681,0] := 3949.0, [682,0] := 3956.0, [683,0] := 3956.0, [684,0] := 3952.0, [685,0] := 3952.0, [686,0] := 3952.0, [687,0] := 3952.0, [688,0] := 3952.0, [689,0] := 3952.0, [690,0] := 3952.0, [691,0] := 3952.0, [692,0] := 3952.0, [693,0] := 3952.0, [694,0] := 3952.0, [695,0] := 3952.0, [696,0] := 3951.0, [697,0] := 3951.0, [698,0] := 3951.0, [699,0] := 3951.0, [700,0] := 3954.0, [701,0] := 3954.0, [702,0] := 3954.0, [703,0] := 3954.0, [704,0] := 3954.0, [705,0] := 3954.0, [706,0] := 3948.0, [707,0] := 3948.0, [708,0] := 3960.0, [709,0] := 3960.0, [710,0] := 3960.0, [711,0] := 3960.0, [712,0] := 3960.0, [713,0] := 3947.0, [714,0] := 3947.0, [715,0] := 3947.0, [716,0] := 3947.0, [717,0] := 3955.0, [718,0] := 3955.0, [719,0] := 3955.0, [720,0] := 3955.0, [721,0] := 3955.0, [722,0] := 3955.0, [723,0] := 3952.0, [724,0] := 3952.0,
        [725,0] := 3952.0, [726,0] := 3952.0, [727,0] := 3952.0, [728,0] := 3952.0, [729,0] := 3952.0, [730,0] := 3952.0, [731,0] := 3952.0, [732,0] := 3952.0, [733,0] := 3952.0, [734,0] := 3959.0, [735,0] := 3959.0, [736,0] := 3959.0, [737,0] := 3959.0, [738,0] := 3959.0, [739,0] := 3959.0, [740,0] := 3959.0, [741,0] := 3959.0, [742,0] := 3956.0, [743,0] := 3956.0, [744,0] := 3956.0, [745,0] := 3956.0, [746,0] := 3956.0, [747,0] := 3956.0, [748,0] := 3956.0, [749,0] := 3944.0, [750,0] := 3944.0, [751,0] := 3944.0, [752,0] := 3944.0, [753,0] := 3953.0, [754,0] := 3953.0, [755,0] := 3953.0, [756,0] := 3953.0, [757,0] := 3953.0, [758,0] := 3953.0, [759,0] := 3945.0, [760,0] := 3945.0, [761,0] := 3945.0, [762,0] := 3945.0, [763,0] := 3945.0, [764,0] := 3945.0, [765,0] := 3945.0, [766,0] := 3945.0, [767,0] := 3945.0, [768,0] := 3945.0, [769,0] := 3945.0, [770,0] := 3947.0, [771,0] := 3947.0, [772,0] := 3947.0, [773,0] := 3947.0, [774,0] := 3947.0, [775,0] := 3948.0, [776,0] := 3948.0, [777,0] := 3948.0, [778,0] := 3948.0, [779,0] := 3948.0, [780,0] := 3948.0, [781,0] := 3948.0, [782,0] := 3955.0, [783,0] := 3955.0, [784,0] := 3955.0,
        [785,0] := 3955.0, [786,0] := 3955.0, [787,0] := 3955.0, [788,0] := 3955.0, [789,0] := 3955.0, [790,0] := 3955.0, [791,0] := 3955.0, [792,0] := 3955.0, [793,0] := 3955.0, [794,0] := 3944.0, [795,0] := 3944.0, [796,0] := 3944.0, [797,0] := 3944.0, [798,0] := 3944.0, [799,0] := 3944.0, [800,0] := 3956.0, [801,0] := 3956.0, [802,0] := 3956.0, [803,0] := 3952.0, [804,0] := 3948.0, [805,0] := 3948.0, [806,0] := 3948.0, [807,0] := 3948.0, [808,0] := 3948.0, [809,0] := 3954.0, [810,0] := 3954.0, [811,0] := 3954.0, [812,0] := 3954.0, [813,0] := 3952.0, [814,0] := 3952.0, [815,0] := 3952.0, [816,0] := 3952.0, [817,0] := 3952.0, [818,0] := 3952.0, [819,0] := 3952.0, [820,0] := 3952.0, [821,0] := 3952.0, [822,0] := 3952.0, [823,0] := 3952.0, [824,0] := 3952.0, [825,0] := 3952.0, [826,0] := 3952.0, [827,0] := 3952.0, [828,0] := 3952.0, [829,0] := 3952.0, [830,0] := 3952.0, [831,0] := 3961.0, [832,0] := 3961.0, [833,0] := 3945.0, [834,0] := 3945.0, [835,0] := 3945.0, [836,0] := 3945.0, [837,0] := 3953.0, [838,0] := 3953.0, [839,0] := 3953.0, [840,0] := 3953.0, [841,0] := 3953.0, [842,0] := 3953.0, [843,0] := 3945.0, [844,0] := 3945.0,
        [845,0] := 3953.0, [846,0] := 3953.0, [847,0] := 3953.0, [848,0] := 3953.0, [849,0] := 3953.0, [850,0] := 3953.0, [851,0] := 3953.0, [852,0] := 3953.0, [853,0] := 3953.0, [854,0] := 3953.0, [855,0] := 3953.0, [856,0] := 3953.0, [857,0] := 3953.0, [858,0] := 3953.0, [859,0] := 3953.0, [860,0] := 3953.0, [861,0] := 3953.0, [862,0] := 3949.0, [863,0] := 3949.0, [864,0] := 3949.0, [865,0] := 3949.0, [866,0] := 3958.0, [867,0] := 3958.0, [868,0] := 3958.0, [869,0] := 3958.0, [870,0] := 3958.0, [871,0] := 3958.0, [872,0] := 3958.0, [873,0] := 3958.0, [874,0] := 3958.0, [875,0] := 3958.0, [876,0] := 3958.0, [877,0] := 3958.0, [878,0] := 3956.0, [879,0] := 3956.0, [880,0] := 3956.0, [881,0] := 3956.0, [882,0] := 3956.0, [883,0] := 3956.0, [884,0] := 3956.0, [885,0] := 3956.0, [886,0] := 3956.0, [887,0] := 3956.0, [888,0] := 3956.0, [889,0] := 3956.0, [890,0] := 3956.0, [891,0] := 3955.0, [892,0] := 3955.0, [893,0] := 3955.0, [894,0] := 3955.0, [895,0] := 3955.0, [896,0] := 3955.0, [897,0] := 3955.0, [898,0] := 3955.0, [899,0] := 3955.0, [900,0] := 3955.0, [901,0] := 3955.0, [902,0] := 3955.0, [903,0] := 3955.0, [904,0] := 3955.0,
        [905,0] := 3955.0, [906,0] := 3955.0, [907,0] := 3955.0, [908,0] := 3948.0, [909,0] := 3948.0, [910,0] := 3951.0, [911,0] := 3951.0, [912,0] := 3951.0, [913,0] := 3951.0, [914,0] := 3943.0, [915,0] := 3943.0, [916,0] := 3943.0, [917,0] := 3943.0, [918,0] := 3951.0, [919,0] := 3951.0, [920,0] := 3954.0, [921,0] := 3954.0, [922,0] := 3954.0, [923,0] := 3954.0, [924,0] := 3954.0, [925,0] := 3954.0, [926,0] := 3954.0, [927,0] := 3949.0, [928,0] := 3949.0, [929,0] := 3949.0, [930,0] := 3949.0, [931,0] := 3949.0, [932,0] := 3949.0, [933,0] := 3949.0, [934,0] := 3949.0, [935,0] := 3949.0, [936,0] := 3949.0, [937,0] := 3949.0, [938,0] := 3949.0, [939,0] := 3943.0, [940,0] := 3943.0, [941,0] := 3943.0, [942,0] := 3943.0, [943,0] := 3943.0, [944,0] := 3943.0, [945,0] := 3943.0, [946,0] := 3943.0, [947,0] := 3943.0, [948,0] := 3948.0, [949,0] := 3948.0, [950,0] := 3948.0, [951,0] := 3954.0, [952,0] := 3954.0, [953,0] := 3954.0, [954,0] := 3954.0, [955,0] := 3954.0, [956,0] := 3954.0, [957,0] := 3954.0, [958,0] := 3954.0, [959,0] := 3954.0, [960,0] := 3951.0, [961,0] := 3951.0, [962,0] := 3951.0, [963,0] := 3951.0, [964,0] := 3951.0,
        [965,0] := 3951.0, [966,0] := 3951.0, [967,0] := 3951.0, [968,0] := 3951.0, [969,0] := 3951.0, [970,0] := 3951.0, [971,0] := 3951.0, [972,0] := 3951.0, [973,0] := 3951.0, [974,0] := 3951.0, [975,0] := 3955.0, [976,0] := 3955.0, [977,0] := 3955.0, [978,0] := 3955.0, [979,0] := 3955.0, [980,0] := 3959.0, [981,0] := 3959.0, [982,0] := 3959.0, [983,0] := 3959.0, [984,0] := 3959.0, [985,0] := 3959.0, [986,0] := 3959.0, [987,0] := 3959.0, [988,0] := 3959.0, [989,0] := 3953.0, [990,0] := 3953.0, [991,0] := 3953.0, [992,0] := 3953.0, [993,0] := 3953.0);
   _edbHalfWindowFilterSize : DINT := 5;
   _edbIdx : DINT := 783;
   _edbParUseWeigths : BOOL;
   _edbParWeights : REAL[31];
   _edbPressArrFiltered : REAL[1000,2] := ([5,0] := 984.0, [6,0] := 984.0, [7,0] := 984.0, [8,0] := 984.0, [9,0] := 984.0, [10,0] := 984.0, [11,0] := 983.0, [12,0] := 983.0, [13,0] := 984.0, [14,0] := 984.0, [15,0] := 984.0, [16,0] := 984.0, [17,0] := 984.0, [18,0] := 984.0, [19,0] := 984.0, [20,0] := 984.0, [21,0] := 984.0, [22,0] := 984.0, [23,0] := 984.0, [24,0] := 984.0, [25,0] := 984.0, [26,0] := 984.0, [27,0] := 984.0, [28,0] := 984.0, [29,0] := 984.0, [30,0] := 984.0, [31,0] := 984.0, [32,0] := 984.0, [33,0] := 984.0, [34,0] := 984.0, [35,0] := 984.0, [36,0] := 984.0, [37,0] := 984.0, [38,0] := 984.0, [39,0] := 984.0, [40,0] := 984.0, [41,0] := 984.0, [42,0] := 984.0, [43,0] := 984.0, [44,0] := 984.0, [45,0] := 984.0, [46,0] := 984.0, [47,0] := 984.0, [48,0] := 984.0, [49,0] := 984.0, [50,0] := 984.0, [51,0] := 984.0, [52,0] := 984.0, [53,0] := 984.0, [54,0] := 984.0, [55,0] := 984.0, [56,0] := 984.0, [57,0] := 984.0, [58,0] := 984.0, [59,0] := 984.0, [60,0] := 984.0, [61,0] := 984.0, [62,0] := 984.0, [63,0] := 984.0, [64,0] := 984.0,
        [65,0] := 984.0, [66,0] := 984.0, [67,0] := 984.0, [68,0] := 984.0, [69,0] := 984.0, [70,0] := 984.0, [71,0] := 984.0, [72,0] := 984.0, [73,0] := 984.0, [74,0] := 984.0, [75,0] := 984.0, [76,0] := 984.0, [77,0] := 984.0, [78,0] := 984.0, [79,0] := 984.0, [80,0] := 984.0, [81,0] := 984.0, [82,0] := 984.0, [83,0] := 984.0, [84,0] := 984.0, [85,0] := 984.0, [86,0] := 984.0, [87,0] := 984.0, [88,0] := 984.0, [89,0] := 984.0, [90,0] := 984.0, [91,0] := 984.0, [92,0] := 984.0, [93,0] := 984.0, [94,0] := 984.0, [95,0] := 984.0, [96,0] := 984.0, [97,0] := 984.0, [98,0] := 984.0, [99,0] := 984.0, [100,0] := 984.0, [101,0] := 984.0, [102,0] := 984.0, [103,0] := 984.0, [104,0] := 984.0, [105,0] := 984.0, [106,0] := 984.0, [107,0] := 984.0, [108,0] := 984.0, [109,0] := 984.0, [110,0] := 984.0, [111,0] := 984.0, [112,0] := 984.0, [113,0] := 984.0, [114,0] := 984.0, [115,0] := 984.0, [116,0] := 984.0, [117,0] := 984.0, [118,0] := 984.0, [119,0] := 984.0, [120,0] := 984.0, [121,0] := 984.0, [122,0] := 984.0, [123,0] := 984.0, [124,0] := 984.0,
        [125,0] := 984.0, [126,0] := 984.0, [127,0] := 984.0, [128,0] := 984.0, [129,0] := 983.0, [130,0] := 983.0, [131,0] := 984.0, [132,0] := 984.0, [133,0] := 984.0, [134,0] := 984.0, [135,0] := 984.0, [136,0] := 984.0, [137,0] := 984.0, [138,0] := 984.0, [139,0] := 984.0, [140,0] := 984.0, [141,0] := 984.0, [142,0] := 984.0, [143,0] := 984.0, [144,0] := 984.0, [145,0] := 984.0, [146,0] := 983.0, [147,0] := 983.0, [148,0] := 984.0, [149,0] := 984.0, [150,0] := 984.0, [151,0] := 984.0, [152,0] := 984.0, [153,0] := 983.0, [154,0] := 983.0, [155,0] := 984.0, [156,0] := 984.0, [157,0] := 984.0, [158,0] := 984.0, [159,0] := 984.0, [160,0] := 984.0, [161,0] := 984.0, [162,0] := 984.0, [163,0] := 984.0, [164,0] := 984.0, [165,0] := 984.0, [166,0] := 984.0, [167,0] := 984.0, [168,0] := 984.0, [169,0] := 984.0, [170,0] := 983.0, [171,0] := 983.0, [172,0] := 984.0, [173,0] := 984.0, [174,0] := 984.0, [175,0] := 984.0, [176,0] := 984.0, [177,0] := 984.0, [178,0] := 984.0, [179,0] := 984.0, [180,0] := 984.0, [181,0] := 984.0, [182,0] := 984.0, [183,0] := 984.0, [184,0] := 984.0,
        [185,0] := 984.0, [186,0] := 984.0, [187,0] := 984.0, [188,0] := 984.0, [189,0] := 984.0, [190,0] := 984.0, [191,0] := 984.0, [192,0] := 984.0, [193,0] := 984.0, [194,0] := 984.0, [195,0] := 984.0, [196,0] := 984.0, [197,0] := 984.0, [198,0] := 984.0, [199,0] := 984.0, [200,0] := 984.0, [201,0] := 984.0, [202,0] := 984.0, [203,0] := 984.0, [204,0] := 984.0, [205,0] := 984.0, [206,0] := 984.0, [207,0] := 984.0, [208,0] := 984.0, [209,0] := 984.0, [210,0] := 984.0, [211,0] := 984.0, [212,0] := 984.0, [213,0] := 984.0, [214,0] := 984.0, [215,0] := 984.0, [216,0] := 984.0, [217,0] := 984.0, [218,0] := 984.0, [219,0] := 984.0, [220,0] := 984.0, [221,0] := 984.0, [222,0] := 984.0, [223,0] := 984.0, [224,0] := 984.0, [225,0] := 984.0, [226,0] := 984.0, [227,0] := 984.0, [228,0] := 984.0, [229,0] := 984.0, [230,0] := 984.0, [231,0] := 984.0, [232,0] := 984.0, [233,0] := 984.0, [234,0] := 984.0, [235,0] := 984.0, [236,0] := 984.0, [237,0] := 984.0, [238,0] := 984.0, [239,0] := 984.0, [240,0] := 984.0, [241,0] := 984.0, [242,0] := 984.0, [243,0] := 984.0, [244,0] := 984.0,
        [245,0] := 984.0, [246,0] := 984.0, [247,0] := 984.0, [248,0] := 984.0, [249,0] := 984.0, [250,0] := 984.0, [251,0] := 984.0, [252,0] := 984.0, [253,0] := 984.0, [254,0] := 984.0, [255,0] := 984.0, [256,0] := 984.0, [257,0] := 984.0, [258,0] := 984.0, [259,0] := 984.0, [260,0] := 984.0, [261,0] := 984.0, [262,0] := 984.0, [263,0] := 984.0, [264,0] := 984.0, [265,0] := 984.0, [266,0] := 984.0, [267,0] := 984.0, [268,0] := 984.0, [269,0] := 984.0, [270,0] := 984.0, [271,0] := 983.0, [272,0] := 983.0, [273,0] := 983.0, [274,0] := 983.0, [275,0] := 984.0, [276,0] := 984.0, [277,0] := 984.0, [278,0] := 984.0, [279,0] := 983.0, [280,0] := 983.0, [281,0] := 983.0, [282,0] := 984.0, [283,0] := 984.0, [284,0] := 984.0, [285,0] := 984.0, [286,0] := 984.0, [287,0] := 984.0, [288,0] := 983.0, [289,0] := 983.0, [290,0] := 984.0, [291,0] := 984.0, [292,0] := 984.0, [293,0] := 984.0, [294,0] := 984.0, [295,0] := 984.0, [296,0] := 984.0, [297,0] := 984.0, [298,0] := 984.0, [299,0] := 984.0, [300,0] := 984.0, [301,0] := 984.0, [302,0] := 984.0, [303,0] := 984.0, [304,0] := 984.0,
        [305,0] := 984.0, [306,0] := 984.0, [307,0] := 984.0, [308,0] := 984.0, [309,0] := 984.0, [310,0] := 984.0, [311,0] := 984.0, [312,0] := 984.0, [313,0] := 984.0, [314,0] := 984.0, [315,0] := 984.0, [316,0] := 984.0, [317,0] := 984.0, [318,0] := 984.0, [319,0] := 984.0, [320,0] := 984.0, [321,0] := 984.0, [322,0] := 984.0, [323,0] := 984.0, [324,0] := 984.0, [325,0] := 984.0, [326,0] := 984.0, [327,0] := 984.0, [328,0] := 984.0, [329,0] := 984.0, [330,0] := 984.0, [331,0] := 984.0, [332,0] := 984.0, [333,0] := 984.0, [334,0] := 984.0, [335,0] := 984.0, [336,0] := 984.0, [337,0] := 984.0, [338,0] := 984.0, [339,0] := 984.0, [340,0] := 984.0, [341,0] := 984.0, [342,0] := 984.0, [343,0] := 984.0, [344,0] := 984.0, [345,0] := 984.0, [346,0] := 984.0, [347,0] := 984.0, [348,0] := 984.0, [349,0] := 984.0, [350,0] := 984.0, [351,0] := 984.0, [352,0] := 984.0, [353,0] := 984.0, [354,0] := 984.0, [355,0] := 984.0, [356,0] := 984.0, [357,0] := 984.0, [358,0] := 984.0, [359,0] := 984.0, [360,0] := 984.0, [361,0] := 984.0, [362,0] := 984.0, [363,0] := 984.0, [364,0] := 984.0,
        [365,0] := 984.0, [366,0] := 984.0, [367,0] := 984.0, [368,0] := 984.0, [369,0] := 984.0, [370,0] := 984.0, [371,0] := 984.0, [372,0] := 984.0, [373,0] := 984.0, [374,0] := 984.0, [375,0] := 984.0, [376,0] := 984.0, [377,0] := 984.0, [378,0] := 984.0, [379,0] := 984.0, [380,0] := 984.0, [381,0] := 984.0, [382,0] := 984.0, [383,0] := 984.0, [384,0] := 984.0, [385,0] := 984.0, [386,0] := 984.0, [387,0] := 984.0, [388,0] := 984.0, [389,0] := 984.0, [390,0] := 984.0, [391,0] := 984.0, [392,0] := 984.0, [393,0] := 984.0, [394,0] := 984.0, [395,0] := 984.0, [396,0] := 984.0, [397,0] := 984.0, [398,0] := 984.0, [399,0] := 984.0, [400,0] := 984.0, [401,0] := 984.0, [402,0] := 984.0, [403,0] := 984.0, [404,0] := 984.0, [405,0] := 984.0, [406,0] := 984.0, [407,0] := 984.0, [408,0] := 984.0, [409,0] := 984.0, [410,0] := 984.0, [411,0] := 984.0, [412,0] := 984.0, [413,0] := 984.0, [414,0] := 984.0, [415,0] := 984.0, [416,0] := 984.0, [417,0] := 984.0, [418,0] := 984.0, [419,0] := 984.0, [420,0] := 984.0, [421,0] := 984.0, [422,0] := 984.0, [423,0] := 984.0, [424,0] := 984.0,
        [425,0] := 984.0, [426,0] := 984.0, [427,0] := 984.0, [428,0] := 984.0, [429,0] := 984.0, [430,0] := 984.0, [431,0] := 984.0, [432,0] := 984.0, [433,0] := 984.0, [434,0] := 984.0, [435,0] := 984.0, [436,0] := 984.0, [437,0] := 984.0, [438,0] := 984.0, [439,0] := 984.0, [440,0] := 984.0, [441,0] := 984.0, [442,0] := 984.0, [443,0] := 984.0, [444,0] := 984.0, [445,0] := 984.0, [446,0] := 984.0, [447,0] := 983.0, [448,0] := 983.0, [449,0] := 984.0, [450,0] := 984.0, [451,0] := 984.0, [452,0] := 984.0, [453,0] := 984.0, [454,0] := 983.0, [455,0] := 983.0, [456,0] := 984.0, [457,0] := 984.0, [458,0] := 984.0, [459,0] := 984.0, [460,0] := 984.0, [461,0] := 984.0, [462,0] := 983.0, [463,0] := 983.0, [464,0] := 983.0, [465,0] := 984.0, [466,0] := 984.0, [467,0] := 984.0, [468,0] := 984.0, [469,0] := 983.0, [470,0] := 983.0, [471,0] := 983.0, [472,0] := 983.0, [473,0] := 984.0, [474,0] := 984.0, [475,0] := 984.0, [476,0] := 984.0, [477,0] := 984.0, [478,0] := 984.0, [479,0] := 984.0, [480,0] := 984.0, [481,0] := 984.0, [482,0] := 984.0, [483,0] := 984.0, [484,0] := 984.0,
        [485,0] := 984.0, [486,0] := 984.0, [487,0] := 984.0, [488,0] := 984.0, [489,0] := 984.0, [490,0] := 984.0, [491,0] := 984.0, [492,0] := 984.0, [493,0] := 984.0, [494,0] := 984.0, [495,0] := 984.0, [496,0] := 984.0, [497,0] := 984.0, [498,0] := 984.0, [499,0] := 984.0, [500,0] := 984.0, [501,0] := 984.0, [502,0] := 984.0, [503,0] := 984.0, [504,0] := 984.0, [505,0] := 984.0, [506,0] := 984.0, [507,0] := 984.0, [508,0] := 984.0, [509,0] := 984.0, [510,0] := 984.0, [511,0] := 984.0, [512,0] := 984.0, [513,0] := 984.0, [514,0] := 984.0, [515,0] := 984.0, [516,0] := 984.0, [517,0] := 984.0, [518,0] := 984.0, [519,0] := 984.0, [520,0] := 984.0, [521,0] := 984.0, [522,0] := 984.0, [523,0] := 984.0, [524,0] := 984.0, [525,0] := 984.0, [526,0] := 984.0, [527,0] := 984.0, [528,0] := 984.0, [529,0] := 984.0, [530,0] := 984.0, [531,0] := 984.0, [532,0] := 984.0, [533,0] := 984.0, [534,0] := 984.0, [535,0] := 984.0, [536,0] := 984.0, [537,0] := 984.0, [538,0] := 984.0, [539,0] := 984.0, [540,0] := 984.0, [541,0] := 984.0, [542,0] := 984.0, [543,0] := 984.0, [544,0] := 984.0,
        [545,0] := 984.0, [546,0] := 984.0, [547,0] := 984.0, [548,0] := 983.0, [549,0] := 983.0, [550,0] := 984.0, [551,0] := 984.0, [552,0] := 984.0, [553,0] := 984.0, [554,0] := 984.0, [555,0] := 984.0, [556,0] := 984.0, [557,0] := 984.0, [558,0] := 984.0, [559,0] := 984.0, [560,0] := 984.0, [561,0] := 984.0, [562,0] := 984.0, [563,0] := 984.0, [564,0] := 984.0, [565,0] := 984.0, [566,0] := 984.0, [567,0] := 984.0, [568,0] := 984.0, [569,0] := 984.0, [570,0] := 984.0, [571,0] := 984.0, [572,0] := 984.0, [573,0] := 984.0, [574,0] := 984.0, [575,0] := 984.0, [576,0] := 984.0, [577,0] := 984.0, [578,0] := 984.0, [579,0] := 984.0, [580,0] := 984.0, [581,0] := 984.0, [582,0] := 984.0, [583,0] := 984.0, [584,0] := 984.0, [585,0] := 984.0, [586,0] := 984.0, [587,0] := 984.0, [588,0] := 984.0, [589,0] := 984.0, [590,0] := 984.0, [591,0] := 984.0, [592,0] := 984.0, [593,0] := 984.0, [594,0] := 984.0, [595,0] := 984.0, [596,0] := 984.0, [597,0] := 984.0, [598,0] := 984.0, [599,0] := 984.0, [600,0] := 984.0, [601,0] := 984.0, [602,0] := 984.0, [603,0] := 984.0, [604,0] := 984.0,
        [605,0] := 984.0, [606,0] := 984.0, [607,0] := 984.0, [608,0] := 984.0, [609,0] := 984.0, [610,0] := 984.0, [611,0] := 984.0, [612,0] := 984.0, [613,0] := 984.0, [614,0] := 984.0, [615,0] := 984.0, [616,0] := 984.0, [617,0] := 984.0, [618,0] := 984.0, [619,0] := 984.0, [620,0] := 984.0, [621,0] := 984.0, [622,0] := 984.0, [623,0] := 984.0, [624,0] := 984.0, [625,0] := 984.0, [626,0] := 984.0, [627,0] := 984.0, [628,0] := 984.0, [629,0] := 983.0, [630,0] := 983.0, [631,0] := 984.0, [632,0] := 984.0, [633,0] := 984.0, [634,0] := 984.0, [635,0] := 983.0, [636,0] := 983.0, [637,0] := 983.0, [638,0] := 983.0, [639,0] := 984.0, [640,0] := 984.0, [641,0] := 984.0, [642,0] := 984.0, [643,0] := 984.0, [644,0] := 984.0, [645,0] := 984.0, [646,0] := 984.0, [647,0] := 984.0, [648,0] := 984.0, [649,0] := 984.0, [650,0] := 984.0, [651,0] := 984.0, [652,0] := 984.0, [653,0] := 984.0, [654,0] := 984.0, [655,0] := 984.0, [656,0] := 984.0, [657,0] := 984.0, [658,0] := 984.0, [659,0] := 984.0, [660,0] := 984.0, [661,0] := 984.0, [662,0] := 984.0, [663,0] := 984.0, [664,0] := 984.0,
        [665,0] := 984.0, [666,0] := 984.0, [667,0] := 984.0, [668,0] := 984.0, [669,0] := 984.0, [670,0] := 984.0, [671,0] := 984.0, [672,0] := 984.0, [673,0] := 984.0, [674,0] := 984.0, [675,0] := 984.0, [676,0] := 984.0, [677,0] := 984.0, [678,0] := 984.0, [679,0] := 984.0, [680,0] := 984.0, [681,0] := 984.0, [682,0] := 984.0, [683,0] := 984.0, [684,0] := 984.0, [685,0] := 984.0, [686,0] := 984.0, [687,0] := 984.0, [688,0] := 984.0, [689,0] := 984.0, [690,0] := 984.0, [691,0] := 984.0, [692,0] := 984.0, [693,0] := 984.0, [694,0] := 984.0, [695,0] := 984.0, [696,0] := 984.0, [697,0] := 984.0, [698,0] := 984.0, [699,0] := 984.0, [700,0] := 984.0, [701,0] := 984.0, [702,0] := 984.0, [703,0] := 984.0, [704,0] := 984.0, [705,0] := 984.0, [706,0] := 984.0, [707,0] := 984.0, [708,0] := 984.0, [709,0] := 984.0, [710,0] := 984.0, [711,0] := 984.0, [712,0] := 984.0, [713,0] := 984.0, [714,0] := 984.0, [715,0] := 984.0, [716,0] := 984.0, [717,0] := 984.0, [718,0] := 984.0, [719,0] := 984.0, [720,0] := 984.0, [721,0] := 984.0, [722,0] := 984.0, [723,0] := 984.0, [724,0] := 984.0,
        [725,0] := 984.0, [726,0] := 984.0, [727,0] := 984.0, [728,0] := 984.0, [729,0] := 984.0, [730,0] := 984.0, [731,0] := 983.0, [732,0] := 983.0, [733,0] := 984.0, [734,0] := 984.0, [735,0] := 984.0, [736,0] := 984.0, [737,0] := 984.0, [738,0] := 984.0, [739,0] := 984.0, [740,0] := 984.0, [741,0] := 984.0, [742,0] := 984.0, [743,0] := 984.0, [744,0] := 984.0, [745,0] := 984.0, [746,0] := 984.0, [747,0] := 984.0, [748,0] := 984.0, [749,0] := 984.0, [750,0] := 984.0, [751,0] := 984.0, [752,0] := 984.0, [753,0] := 984.0, [754,0] := 984.0, [755,0] := 983.0, [756,0] := 983.0, [757,0] := 984.0, [758,0] := 984.0, [759,0] := 984.0, [760,0] := 984.0, [761,0] := 984.0, [762,0] := 984.0, [763,0] := 984.0, [764,0] := 984.0, [765,0] := 984.0, [766,0] := 984.0, [767,0] := 984.0, [768,0] := 984.0, [769,0] := 984.0, [770,0] := 984.0, [771,0] := 984.0, [772,0] := 984.0, [773,0] := 984.0, [774,0] := 984.0, [775,0] := 984.0, [776,0] := 984.0, [777,0] := 984.0, [778,0] := 984.0, [779,0] := 983.0, [780,0] := 983.0, [781,0] := 984.0, [782,0] := 984.0, [783,0] := 984.0, [784,0] := 984.0,
        [785,0] := 984.0, [786,0] := 984.0, [787,0] := 984.0, [788,0] := 984.0, [789,0] := 984.0, [790,0] := 984.0, [791,0] := 984.0, [792,0] := 984.0, [793,0] := 984.0, [794,0] := 984.0, [795,0] := 984.0, [796,0] := 984.0, [797,0] := 984.0, [798,0] := 984.0, [799,0] := 984.0, [800,0] := 984.0, [801,0] := 984.0, [802,0] := 984.0, [803,0] := 984.0, [804,0] := 984.0, [805,0] := 984.0, [806,0] := 984.0, [807,0] := 984.0, [808,0] := 984.0, [809,0] := 984.0, [810,0] := 984.0, [811,0] := 984.0, [812,0] := 984.0, [813,0] := 984.0, [814,0] := 984.0, [815,0] := 984.0, [816,0] := 984.0, [817,0] := 984.0, [818,0] := 984.0, [819,0] := 984.0, [820,0] := 984.0, [821,0] := 984.0, [822,0] := 984.0, [823,0] := 984.0, [824,0] := 984.0, [825,0] := 984.0, [826,0] := 984.0, [827,0] := 983.0, [828,0] := 983.0, [829,0] := 984.0, [830,0] := 984.0, [831,0] := 984.0, [832,0] := 984.0, [833,0] := 984.0, [834,0] := 984.0, [835,0] := 984.0, [836,0] := 984.0, [837,0] := 984.0, [838,0] := 984.0, [839,0] := 984.0, [840,0] := 984.0, [841,0] := 984.0, [842,0] := 984.0, [843,0] := 984.0, [844,0] := 984.0,
        [845,0] := 984.0, [846,0] := 984.0, [847,0] := 984.0, [848,0] := 984.0, [849,0] := 984.0, [850,0] := 984.0, [851,0] := 984.0, [852,0] := 984.0, [853,0] := 984.0, [854,0] := 984.0, [855,0] := 984.0, [856,0] := 984.0, [857,0] := 984.0, [858,0] := 984.0, [859,0] := 984.0, [860,0] := 984.0, [861,0] := 984.0, [862,0] := 984.0, [863,0] := 984.0, [864,0] := 984.0, [865,0] := 984.0, [866,0] := 984.0, [867,0] := 983.0, [868,0] := 983.0, [869,0] := 984.0, [870,0] := 984.0, [871,0] := 984.0, [872,0] := 984.0, [873,0] := 983.0, [874,0] := 983.0, [875,0] := 983.0, [876,0] := 983.0, [877,0] := 984.0, [878,0] := 984.0, [879,0] := 984.0, [880,0] := 984.0, [881,0] := 984.0, [882,0] := 984.0, [883,0] := 984.0, [884,0] := 984.0, [885,0] := 984.0, [886,0] := 984.0, [887,0] := 984.0, [888,0] := 984.0, [889,0] := 984.0, [890,0] := 984.0, [891,0] := 984.0, [892,0] := 984.0, [893,0] := 984.0, [894,0] := 984.0, [895,0] := 984.0, [896,0] := 984.0, [897,0] := 984.0, [898,0] := 984.0, [899,0] := 984.0, [900,0] := 984.0, [901,0] := 984.0, [902,0] := 984.0, [903,0] := 984.0, [904,0] := 984.0,
        [905,0] := 984.0, [906,0] := 984.0, [907,0] := 984.0, [908,0] := 984.0, [909,0] := 984.0, [910,0] := 984.0, [911,0] := 984.0, [912,0] := 984.0, [913,0] := 984.0, [914,0] := 984.0, [915,0] := 984.0, [916,0] := 984.0, [917,0] := 984.0, [918,0] := 984.0, [919,0] := 984.0, [920,0] := 984.0, [921,0] := 983.0, [922,0] := 983.0, [923,0] := 984.0, [924,0] := 984.0, [925,0] := 984.0, [926,0] := 984.0, [927,0] := 984.0, [928,0] := 984.0, [929,0] := 984.0, [930,0] := 984.0, [931,0] := 984.0, [932,0] := 984.0, [933,0] := 984.0, [934,0] := 984.0, [935,0] := 984.0, [936,0] := 984.0, [937,0] := 984.0, [938,0] := 984.0, [939,0] := 984.0, [940,0] := 984.0, [941,0] := 984.0, [942,0] := 984.0, [943,0] := 984.0, [944,0] := 984.0, [945,0] := 983.0, [946,0] := 983.0, [947,0] := 984.0, [948,0] := 984.0, [949,0] := 984.0, [950,0] := 984.0, [951,0] := 984.0, [952,0] := 984.0, [953,0] := 984.0, [954,0] := 984.0, [955,0] := 984.0, [956,0] := 984.0, [957,0] := 984.0, [958,0] := 984.0, [959,0] := 984.0, [960,0] := 984.0, [961,0] := 984.0, [962,0] := 984.0, [963,0] := 984.0, [964,0] := 984.0,
        [965,0] := 984.0, [966,0] := 984.0, [967,0] := 984.0, [968,0] := 984.0, [969,0] := 984.0, [970,0] := 984.0, [971,0] := 984.0, [972,0] := 984.0, [973,0] := 984.0, [974,0] := 984.0, [975,0] := 984.0, [976,0] := 984.0, [977,0] := 984.0, [978,0] := 984.0, [979,0] := 984.0, [980,0] := 984.0, [981,0] := 984.0, [982,0] := 984.0, [983,0] := 984.0, [984,0] := 984.0, [985,0] := 984.0, [986,0] := 984.0, [987,0] := 985.0, [988,0] := 985.0, [989,0] := 985.0, [990,0] := 985.0, [991,0] := 984.0, [992,0] := 984.0, [993,0] := 984.0);
   _edbTypeOfFilter : DINT;
   _endPosition : DINT;
   _endPositionOld : DINT;
   _EndSendPosition : DINT;
   _i : DINT := 1000;
   _J : INT := 196;
   _n : DINT := 412;
   _PointAfterEnd : DINT := 30;
   _StartPointBerfore : DINT := 30;
   _StartPosition : DINT;
   _StartpositionOld : DINT;
   _T : DINT;
   _z : DINT := 51;
   ActiveinspTimeinMS : REAL := 1200.0;
   AirConstantFlow : REAL := 68.35443;
   AirDown : CAM_PROFILE[1010] := ([0].Status := 2, [1].Status := 2, [2].Status := 2, [3].Status := 2, [4].Status := 2, [5].Status := 2, [6].Status := 2, [7].Status := 2, [8].Status := 2, [9].Status := 2, [10].Status := 2, [11].Status := 2, [12].Status := 2, [13].Status := 2, [14].Status := 2, [15].Status := 2, [16].Status := 2, [17].Status := 2, [18].Status := 2, [19].Status := 2, [20].Status := 2, [21].Status := 2, [22].Status := 2, [23].Status := 2, [24].Status := 2, [25].Status := 2, [26].Status := 2, [27].Status := 2, [28].Status := 2, [29].Status := 2, [30].Status := 2, [31].Status := 2, [32].Status := 2, [33].Status := 2, [34].Status := 2, [35].Status := 2, [36].Status := 2, [37].Status := 2, [38].Status := 2, [39].Status := 2, [40].Status := 2, [41].Status := 2, [42].Status := 2, [43].Status := 2, [44].Status := 2, [45].Status := 2, [46].Status := 2, [47].Status := 2, [48].Status := 2, [49].Status := 2, [50].Status := 2, [51].Status := 2, [52].Status := 2, [53].Status := 2, [54].Status := 2, [55].Status := 2, [56].Status := 2, [57].Status := 2, [58].Status := 2, [59].Status := 2,
        [60].Status := 2, [61].Status := 2, [62].Status := 2, [63].Status := 2, [64].Status := 2, [65].Status := 2, [66].Status := 2, [67].Status := 2, [68].Status := 2, [69].Status := 2, [70].Status := 2, [71].Status := 2, [72].Status := 2, [73].Status := 2, [74].Status := 2, [75].Status := 2, [76].Status := 2, [77].Status := 2, [78].Status := 2, [79].Status := 2, [80].Status := 2, [81].Status := 2, [82].Status := 2, [83].Status := 2, [84].Status := 2, [85].Status := 2, [86].Status := 2, [87].Status := 2, [88].Status := 2, [89].Status := 2, [90].Status := 2, [91].Status := 2, [92].Status := 2, [93].Status := 2, [94].Status := 2, [95].Status := 2, [96].Status := 2, [97].Status := 2, [98].Status := 2, [99].Status := 2, [100].Status := 2, [101].Status := 2, [102].Status := 2, [103].Status := 2, [104].Status := 2, [105].Status := 2, [106].Status := 2, [107].Status := 2, [108].Status := 2, [109].Status := 2, [110].Status := 2, [111].Status := 2, [112].Status := 2, [113].Status := 2, [114].Status := 2, [115].Status := 2, [116].Status := 2, [117].Status := 2, [118].Status := 2, [119].Status := 2,
        [120].Status := 2, [121].Status := 2, [122].Status := 2, [123].Status := 2, [124].Status := 2, [125].Status := 2, [126].Status := 2, [127].Status := 2, [128].Status := 2, [129].Status := 2, [130].Status := 2, [131].Status := 2, [132].Status := 2, [133].Status := 2, [134].Status := 2, [135].Status := 2, [136].Status := 2, [137].Status := 2, [138].Status := 2, [139].Status := 2, [140].Status := 2, [141].Status := 2, [142].Status := 2, [143].Status := 2, [144].Status := 2, [145].Status := 2, [146].Status := 2, [147].Status := 2, [148].Status := 2, [149].Status := 2, [150].Status := 2, [151].Status := 2, [152].Status := 2, [153].Status := 2, [154].Status := 2, [155].Status := 2, [156].Status := 2, [157].Status := 2, [158].Status := 2, [159].Status := 2, [160].Status := 2, [161].Status := 2, [162].Status := 2, [163].Status := 2, [164].Status := 2, [165].Status := 2, [166].Status := 2, [167].Status := 2, [168].Status := 2, [169].Status := 2, [170].Status := 2, [171].Status := 2, [172].Status := 2, [173].Status := 2, [174].Status := 2, [175].Status := 2, [176].Status := 2, [177].Status := 2, [178].Status := 2, [179].Status := 2,
        [180].Status := 2, [181].Status := 2, [182].Status := 2, [183].Status := 2, [184].Status := 2, [185].Status := 2, [186].Status := 2, [187].Status := 2, [188].Status := 2, [189].Status := 2, [190].Status := 2, [191].Status := 2, [192].Status := 2, [193].Status := 2, [194].Status := 2, [195].Status := 2, [196].Status := 2, [197].Status := 2, [198].Status := 2, [199].Status := 2, [200].Status := 2, [201].Status := 2, [202].Status := 2, [203].Status := 2, [204].Status := 2, [205].Status := 2, [206].Status := 2, [207].Status := 2, [208].Status := 2, [209].Status := 2, [210].Status := 2, [211].Status := 2, [212].Status := 2, [213].Status := 2, [214].Status := 2, [215].Status := 2, [216].Status := 2, [217].Status := 2, [218].Status := 2, [219].Status := 2, [220].Status := 2, [221].Status := 2, [222].Status := 2, [223].Status := 2, [224].Status := 2, [225].Status := 2, [226].Status := 2, [227].Status := 2, [228].Status := 2, [229].Status := 2, [230].Status := 2, [231].Status := 2, [232].Status := 2, [233].Status := 2, [234].Status := 2, [235].Status := 2, [236].Status := 2, [237].Status := 2, [238].Status := 2, [239].Status := 2,
        [240].Status := 2, [241].Status := 2, [242].Status := 2, [243].Status := 2, [244].Status := 2, [245].Status := 2, [246].Status := 2, [247].Status := 2, [248].Status := 2, [249].Status := 2, [250].Status := 2, [251].Status := 2, [252].Status := 2, [253].Status := 2, [254].Status := 2, [255].Status := 2, [256].Status := 2, [257].Status := 2, [258].Status := 2, [259].Status := 2, [260].Status := 2, [261].Status := 2, [262].Status := 2, [263].Status := 2, [264].Status := 2, [265].Status := 2, [266].Status := 2, [267].Status := 2, [268].Status := 2, [269].Status := 2, [270].Status := 2, [271].Status := 2, [272].Status := 2, [273].Status := 2, [274].Status := 2, [275].Status := 2, [276].Status := 2, [277].Status := 2, [278].Status := 2, [279].Status := 2, [280].Status := 2, [281].Status := 2, [282].Status := 2, [283].Status := 2, [284].Status := 2, [285].Status := 2, [286].Status := 2, [287].Status := 2, [288].Status := 2, [289].Status := 2, [290].Status := 2, [291].Status := 2, [292].Status := 2, [293].Status := 2, [294].Status := 2, [295].Status := 2, [296].Status := 2, [297].Status := 2, [298].Status := 2, [299].Status := 2,
        [300].Status := 2, [301].Status := 2, [302].Status := 2, [303].Status := 2, [304].Status := 2, [305].Status := 2, [306].Status := 2, [307].Status := 2, [308].Status := 2, [309].Status := 2, [310].Status := 2, [311].Status := 2, [312].Status := 2, [313].Status := 2, [314].Status := 2, [315].Status := 2, [316].Status := 2, [317].Status := 2, [318].Status := 2, [319].Status := 2, [320].Status := 2, [321].Status := 2, [322].Status := 2, [323].Status := 2, [324].Status := 2, [325].Status := 2, [326].Status := 2, [327].Status := 2, [328].Status := 2, [329].Status := 2, [330].Status := 2, [331].Status := 2, [332].Status := 2, [333].Status := 2, [334].Status := 2, [335].Status := 2, [336].Status := 2, [337].Status := 2, [338].Status := 2, [339].Status := 2, [340].Status := 2, [341].Status := 2, [342].Status := 2, [343].Status := 2, [344].Status := 2, [345].Status := 2, [346].Status := 2, [347].Status := 2, [348].Status := 2, [349].Status := 2, [350].Status := 2, [351].Status := 2, [352].Status := 2, [353].Status := 2, [354].Status := 2, [355].Status := 2, [356].Status := 2, [357].Status := 2, [358].Status := 2, [359].Status := 2,
        [360].Status := 2, [361].Status := 2, [362].Status := 2, [363].Status := 2, [364].Status := 2, [365].Status := 2, [366].Status := 2, [367].Status := 2, [368].Status := 2, [369].Status := 2, [370].Status := 2, [371].Status := 2, [372].Status := 2, [373].Status := 2, [374].Status := 2, [375].Status := 2, [376].Status := 2, [377].Status := 2, [378].Status := 2, [379].Status := 2, [380].Status := 2, [381].Status := 2, [382].Status := 2, [383].Status := 2, [384].Status := 2, [385].Status := 2, [386].Status := 2, [387].Status := 2, [388].Status := 2, [389].Status := 2, [390].Status := 2, [391].Status := 2, [392].Status := 2, [393].Status := 2, [394].Status := 2, [395].Status := 2, [396].Status := 2, [397].Status := 2, [398].Status := 2, [399].Status := 2, [400].Status := 2, [401].Status := 2, [402].Status := 2, [403].Status := 2, [404].Status := 2, [405].Status := 2, [406].Status := 2, [407].Status := 2, [408].Status := 2, [409].Status := 2, [410].Status := 2, [411].Status := 2, [412].Status := 2, [413].Status := 2, [414].Status := 2, [415].Status := 2, [416].Status := 2, [417].Status := 2, [418].Status := 2, [419].Status := 2,
        [420].Status := 2, [421].Status := 2, [422].Status := 2, [423].Status := 2, [424].Status := 2, [425].Status := 2, [426].Status := 2, [427].Status := 2, [428].Status := 2, [429].Status := 2, [430].Status := 2, [431].Status := 2, [432].Status := 2, [433].Status := 2, [434].Status := 2, [435].Status := 2, [436].Status := 2, [437].Status := 2, [438].Status := 2, [439].Status := 2, [440].Status := 2, [441].Status := 2, [442].Status := 2, [443].Status := 2, [444].Status := 2, [445].Status := 2, [446].Status := 2, [447].Status := 2, [448].Status := 2, [449].Status := 2, [450].Status := 2, [451].Status := 2, [452].Status := 2, [453].Status := 2, [454].Status := 2, [455].Status := 2, [456].Status := 2, [457].Status := 2, [458].Status := 2, [459].Status := 2, [460].Status := 2, [461].Status := 2, [462].Status := 2, [463].Status := 2, [464].Status := 2, [465].Status := 2, [466].Status := 2, [467].Status := 2, [468].Status := 2, [469].Status := 2, [470].Status := 2, [471].Status := 2, [472].Status := 2, [473].Status := 2, [474].Status := 2, [475].Status := 2, [476].Status := 2, [477].Status := 2, [478].Status := 2, [479].Status := 2,
        [480].Status := 2, [481].Status := 2, [482].Status := 2, [483].Status := 2, [484].Status := 2, [485].Status := 2, [486].Status := 2, [487].Status := 2, [488].Status := 2, [489].Status := 2, [490].Status := 2, [491].Status := 2, [492].Status := 2, [493].Status := 2, [494].Status := 2, [495].Status := 2, [496].Status := 2, [497].Status := 2, [498].Status := 2, [499].Status := 2, [500].Status := 2, [501].Status := 2, [502].Status := 2, [503].Status := 2, [504].Status := 2, [505].Status := 2, [506].Status := 2, [507].Status := 2, [508].Status := 2, [509].Status := 2, [510].Status := 2, [511].Status := 2, [512].Status := 2, [513].Status := 2, [514].Status := 2, [515].Status := 2, [516].Status := 2, [517].Status := 2, [518].Status := 2, [519].Status := 2, [520].Status := 2, [521].Status := 2, [522].Status := 2, [523].Status := 2, [524].Status := 2, [525].Status := 2, [526].Status := 2, [527].Status := 2, [528].Status := 2, [529].Status := 2, [530].Status := 2, [531].Status := 2, [532].Status := 2, [533].Status := 2, [534].Status := 2, [535].Status := 2, [536].Status := 2, [537].Status := 2, [538].Status := 2, [539].Status := 2,
        [540].Status := 2, [541].Status := 2, [542].Status := 2, [543].Status := 2, [544].Status := 2, [545].Status := 2, [546].Status := 2, [547].Status := 2, [548].Status := 2, [549].Status := 2, [550].Status := 2, [551].Status := 2, [552].Status := 2, [553].Status := 2, [554].Status := 2, [555].Status := 2, [556].Status := 2, [557].Status := 2, [558].Status := 2, [559].Status := 2, [560].Status := 2, [561].Status := 2, [562].Status := 2, [563].Status := 2, [564].Status := 2, [565].Status := 2, [566].Status := 2, [567].Status := 2, [568].Status := 2, [569].Status := 2, [570].Status := 2, [571].Status := 2, [572].Status := 2, [573].Status := 2, [574].Status := 2, [575].Status := 2, [576].Status := 2, [577].Status := 2, [578].Status := 2, [579].Status := 2, [580].Status := 2, [581].Status := 2, [582].Status := 2, [583].Status := 2, [584].Status := 2, [585].Status := 2, [586].Status := 2, [587].Status := 2, [588].Status := 2, [589].Status := 2, [590].Status := 2, [591].Status := 2, [592].Status := 2, [593].Status := 2, [594].Status := 2, [595].Status := 2, [596].Status := 2, [597].Status := 2, [598].Status := 2, [599].Status := 2,
        [600].Status := 2, [601].Status := 2, [602].Status := 2, [603].Status := 2, [604].Status := 2, [605].Status := 2, [606].Status := 2, [607].Status := 2, [608].Status := 2, [609].Status := 2, [610].Status := 2, [611].Status := 2, [612].Status := 2, [613].Status := 2, [614].Status := 2, [615].Status := 2, [616].Status := 2, [617].Status := 2, [618].Status := 2, [619].Status := 2, [620].Status := 2, [621].Status := 2, [622].Status := 2, [623].Status := 2, [624].Status := 2, [625].Status := 2, [626].Status := 2, [627].Status := 2, [628].Status := 2, [629].Status := 2, [630].Status := 2, [631].Status := 2, [632].Status := 2, [633].Status := 2, [634].Status := 2, [635].Status := 2, [636].Status := 2, [637].Status := 2, [638].Status := 2, [639].Status := 2, [640].Status := 2, [641].Status := 2, [642].Status := 2, [643].Status := 2, [644].Status := 2, [645].Status := 2, [646].Status := 2, [647].Status := 2, [648].Status := 2, [649].Status := 2, [650].Status := 2, [651].Status := 2, [652].Status := 2, [653].Status := 2, [654].Status := 2, [655].Status := 2, [656].Status := 2, [657].Status := 2, [658].Status := 2, [659].Status := 2,
        [660].Status := 2, [661].Status := 2, [662].Status := 2, [663].Status := 2, [664].Status := 2, [665].Status := 2, [666].Status := 2, [667].Status := 2, [668].Status := 2, [669].Status := 2, [670].Status := 2, [671].Status := 2, [672].Status := 2, [673].Status := 2, [674].Status := 2, [675].Status := 2, [676].Status := 2, [677].Status := 2, [678].Status := 2, [679].Status := 2, [680].Status := 2, [681].Status := 2, [682].Status := 2, [683].Status := 2, [684].Status := 2, [685].Status := 2, [686].Status := 2, [687].Status := 2, [688].Status := 2, [689].Status := 2, [690].Status := 2, [691].Status := 2, [692].Status := 2, [693].Status := 2, [694].Status := 2, [695].Status := 2, [696].Status := 2, [697].Status := 2, [698].Status := 2, [699].Status := 2, [700].Status := 2, [701].Status := 2, [702].Status := 2, [703].Status := 2, [704].Status := 2, [705].Status := 2, [706].Status := 2, [707].Status := 2, [708].Status := 2, [709].Status := 2, [710].Status := 2, [711].Status := 2, [712].Status := 2, [713].Status := 2, [714].Status := 2, [715].Status := 2, [716].Status := 2, [717].Status := 2, [718].Status := 2, [719].Status := 2,
        [720].Status := 2, [721].Status := 2, [722].Status := 2, [723].Status := 2, [724].Status := 2, [725].Status := 2, [726].Status := 2, [727].Status := 2, [728].Status := 2, [729].Status := 2, [730].Status := 2, [731].Status := 2, [732].Status := 2, [733].Status := 2, [734].Status := 2, [735].Status := 2, [736].Status := 2, [737].Status := 2, [738].Status := 2, [739].Status := 2, [740].Status := 2, [741].Status := 2, [742].Status := 2, [743].Status := 2, [744].Status := 2, [745].Status := 2, [746].Status := 2, [747].Status := 2, [748].Status := 2, [749].Status := 2, [750].Status := 2, [751].Status := 2, [752].Status := 2, [753].Status := 2, [754].Status := 2, [755].Status := 2, [756].Status := 2, [757].Status := 2, [758].Status := 2, [759].Status := 2, [760].Status := 2, [761].Status := 2, [762].Status := 2, [763].Status := 2, [764].Status := 2, [765].Status := 2, [766].Status := 2, [767].Status := 2, [768].Status := 2, [769].Status := 2, [770].Status := 2, [771].Status := 2, [772].Status := 2, [773].Status := 2, [774].Status := 2, [775].Status := 2, [776].Status := 2, [777].Status := 2, [778].Status := 2, [779].Status := 2,
        [780].Status := 2, [781].Status := 2, [782].Status := 2, [783].Status := 2, [784].Status := 2, [785].Status := 2, [786].Status := 2, [787].Status := 2, [788].Status := 2, [789].Status := 2, [790].Status := 2, [791].Status := 2, [792].Status := 2, [793].Status := 2, [794].Status := 2, [795].Status := 2, [796].Status := 2, [797].Status := 2, [798].Status := 2, [799].Status := 2, [800].Status := 2, [801].Status := 2, [802].Status := 2, [803].Status := 2, [804].Status := 2, [805].Status := 2, [806].Status := 2, [807].Status := 2, [808].Status := 2, [809].Status := 2, [810].Status := 2, [811].Status := 2, [812].Status := 2, [813].Status := 2, [814].Status := 2, [815].Status := 2, [816].Status := 2, [817].Status := 2, [818].Status := 2, [819].Status := 2, [820].Status := 2, [821].Status := 2, [822].Status := 2, [823].Status := 2, [824].Status := 2, [825].Status := 2, [826].Status := 2, [827].Status := 2, [828].Status := 2, [829].Status := 2, [830].Status := 2, [831].Status := 2, [832].Status := 2, [833].Status := 2, [834].Status := 2, [835].Status := 2, [836].Status := 2, [837].Status := 2, [838].Status := 2, [839].Status := 2,
        [840].Status := 2, [841].Status := 2, [842].Status := 2, [843].Status := 2, [844].Status := 2, [845].Status := 2, [846].Status := 2, [847].Status := 2, [848].Status := 2, [849].Status := 2, [850].Status := 2, [851].Status := 2, [852].Status := 2, [853].Status := 2, [854].Status := 2, [855].Status := 2, [856].Status := 2, [857].Status := 2, [858].Status := 2, [859].Status := 2, [860].Status := 2, [861].Status := 2, [862].Status := 2, [863].Status := 2, [864].Status := 2, [865].Status := 2, [866].Status := 2, [867].Status := 2, [868].Status := 2, [869].Status := 2, [870].Status := 2, [871].Status := 2, [872].Status := 2, [873].Status := 2, [874].Status := 2, [875].Status := 2, [876].Status := 2, [877].Status := 2, [878].Status := 2, [879].Status := 2, [880].Status := 2, [881].Status := 2, [882].Status := 2, [883].Status := 2, [884].Status := 2, [885].Status := 2, [886].Status := 2, [887].Status := 2, [888].Status := 2, [889].Status := 2, [890].Status := 2, [891].Status := 2, [892].Status := 2, [893].Status := 2, [894].Status := 2, [895].Status := 2, [896].Status := 2, [897].Status := 2, [898].Status := 2, [899].Status := 2,
        [900].Status := 2, [901].Status := 2, [902].Status := 2, [903].Status := 2, [904].Status := 2, [905].Status := 2, [906].Status := 2, [907].Status := 2, [908].Status := 2, [909].Status := 2, [910].Status := 2, [911].Status := 2, [912].Status := 2, [913].Status := 2, [914].Status := 2, [915].Status := 2, [916].Status := 2, [917].Status := 2, [918].Status := 2, [919].Status := 2, [920].Status := 2, [921].Status := 2, [922].Status := 2, [923].Status := 2, [924].Status := 2, [925].Status := 2, [926].Status := 2, [927].Status := 2, [928].Status := 2, [929].Status := 2, [930].Status := 2, [931].Status := 2, [932].Status := 2, [933].Status := 2, [934].Status := 2, [935].Status := 2, [936].Status := 2, [937].Status := 2, [938].Status := 2, [939].Status := 2, [940].Status := 2, [941].Status := 2, [942].Status := 2, [943].Status := 2, [944].Status := 2, [945].Status := 2, [946].Status := 2, [947].Status := 2, [948].Status := 2, [949].Status := 2, [950].Status := 2, [951].Status := 2, [952].Status := 2, [953].Status := 2, [954].Status := 2, [955].Status := 2, [956].Status := 2, [957].Status := 2, [958].Status := 2, [959].Status := 2,
        [960].Status := 2, [961].Status := 2, [962].Status := 2, [963].Status := 2, [964].Status := 2, [965].Status := 2, [966].Status := 2, [967].Status := 2, [968].Status := 2, [969].Status := 2, [970].Status := 2, [971].Status := 2, [972].Status := 2, [973].Status := 2, [974].Status := 2, [975].Status := 2, [976].Status := 2, [977].Status := 2, [978].Status := 2, [979].Status := 2, [980].Status := 2, [981].Status := 2, [982].Status := 2, [983].Status := 2, [984].Status := 2, [985].Status := 2, [986].Status := 2, [987].Status := 2, [988].Status := 2, [989].Status := 2, [990].Status := 2, [991].Status := 2, [992].Status := 2, [993].Status := 2, [994].Status := 2, [995].Status := 2, [996].Status := 2, [997].Status := 2, [998].Status := 2, [999].Status := 2, [1000].Status := 2, [1001].Status := 2, [1002].Status := 2);
   AirmADer : REAL;
   AirmAOut : REAL;
   AirmASlope : REAL := 49211.336;
   AirRampFlowIncreasePerAdjust : REAL := 3.4177215;
   AirUp : CAM_PROFILE[1010] := ([0].Status := 2, [1].Status := 2, [2].Status := 2, [3].Status := 2, [4].Status := 2, [5].Status := 2, [6].Status := 2, [7].Status := 2, [8].Status := 2, [9].Status := 2, [10].Status := 2, [11].Status := 2, [12].Status := 2, [13].Status := 2, [14].Status := 2, [15].Status := 2, [16].Status := 2, [17].Status := 2, [18].Status := 2, [19].Status := 2, [20].Status := 2, [21].Status := 2, [22].Status := 2, [23].Status := 2, [24].Status := 2, [25].Status := 2, [26].Status := 2, [27].Status := 2, [28].Status := 2, [29].Status := 2, [30].Status := 2, [31].Status := 2, [32].Status := 2, [33].Status := 2, [34].Status := 2, [35].Status := 2, [36].Status := 2, [37].Status := 2, [38].Status := 2, [39].Status := 2, [40].Status := 2, [41].Status := 2, [42].Status := 2, [43].Status := 2, [44].Status := 2, [45].Status := 2, [46].Status := 2, [47].Status := 2, [48].Status := 2, [49].Status := 2, [50].Status := 2, [51].Status := 2, [52].Status := 2, [53].Status := 2, [54].Status := 2, [55].Status := 2, [56].Status := 2, [57].Status := 2, [58].Status := 2, [59].Status := 2,
        [60].Status := 2, [61].Status := 2, [62].Status := 2, [63].Status := 2, [64].Status := 2, [65].Status := 2, [66].Status := 2, [67].Status := 2, [68].Status := 2, [69].Status := 2, [70].Status := 2, [71].Status := 2, [72].Status := 2, [73].Status := 2, [74].Status := 2, [75].Status := 2, [76].Status := 2, [77].Status := 2, [78].Status := 2, [79].Status := 2, [80].Status := 2, [81].Status := 2, [82].Status := 2, [83].Status := 2, [84].Status := 2, [85].Status := 2, [86].Status := 2, [87].Status := 2, [88].Status := 2, [89].Status := 2, [90].Status := 2, [91].Status := 2, [92].Status := 2, [93].Status := 2, [94].Status := 2, [95].Status := 2, [96].Status := 2, [97].Status := 2, [98].Status := 2, [99].Status := 2, [100].Status := 2, [101].Status := 2, [102].Status := 2, [103].Status := 2, [104].Status := 2, [105].Status := 2, [106].Status := 2, [107].Status := 2, [108].Status := 2, [109].Status := 2, [110].Status := 2, [111].Status := 2, [112].Status := 2, [113].Status := 2, [114].Status := 2, [115].Status := 2, [116].Status := 2, [117].Status := 2, [118].Status := 2, [119].Status := 2,
        [120].Status := 2, [121].Status := 2, [122].Status := 2, [123].Status := 2, [124].Status := 2, [125].Status := 2, [126].Status := 2, [127].Status := 2, [128].Status := 2, [129].Status := 2, [130].Status := 2, [131].Status := 2, [132].Status := 2, [133].Status := 2, [134].Status := 2, [135].Status := 2, [136].Status := 2, [137].Status := 2, [138].Status := 2, [139].Status := 2, [140].Status := 2, [141].Status := 2, [142].Status := 2, [143].Status := 2, [144].Status := 2, [145].Status := 2, [146].Status := 2, [147].Status := 2, [148].Status := 2, [149].Status := 2, [150].Status := 2, [151].Status := 2, [152].Status := 2, [153].Status := 2, [154].Status := 2, [155].Status := 2, [156].Status := 2, [157].Status := 2, [158].Status := 2, [159].Status := 2, [160].Status := 2, [161].Status := 2, [162].Status := 2, [163].Status := 2, [164].Status := 2, [165].Status := 2, [166].Status := 2, [167].Status := 2, [168].Status := 2, [169].Status := 2, [170].Status := 2, [171].Status := 2, [172].Status := 2, [173].Status := 2, [174].Status := 2, [175].Status := 2, [176].Status := 2, [177].Status := 2, [178].Status := 2, [179].Status := 2,
        [180].Status := 2, [181].Status := 2, [182].Status := 2, [183].Status := 2, [184].Status := 2, [185].Status := 2, [186].Status := 2, [187].Status := 2, [188].Status := 2, [189].Status := 2, [190].Status := 2, [191].Status := 2, [192].Status := 2, [193].Status := 2, [194].Status := 2, [195].Status := 2, [196].Status := 2, [197].Status := 2, [198].Status := 2, [199].Status := 2, [200].Status := 2, [201].Status := 2, [202].Status := 2, [203].Status := 2, [204].Status := 2, [205].Status := 2, [206].Status := 2, [207].Status := 2, [208].Status := 2, [209].Status := 2, [210].Status := 2, [211].Status := 2, [212].Status := 2, [213].Status := 2, [214].Status := 2, [215].Status := 2, [216].Status := 2, [217].Status := 2, [218].Status := 2, [219].Status := 2, [220].Status := 2, [221].Status := 2, [222].Status := 2, [223].Status := 2, [224].Status := 2, [225].Status := 2, [226].Status := 2, [227].Status := 2, [228].Status := 2, [229].Status := 2, [230].Status := 2, [231].Status := 2, [232].Status := 2, [233].Status := 2, [234].Status := 2, [235].Status := 2, [236].Status := 2, [237].Status := 2, [238].Status := 2, [239].Status := 2,
        [240].Status := 2, [241].Status := 2, [242].Status := 2, [243].Status := 2, [244].Status := 2, [245].Status := 2, [246].Status := 2, [247].Status := 2, [248].Status := 2, [249].Status := 2, [250].Status := 2, [251].Status := 2, [252].Status := 2, [253].Status := 2, [254].Status := 2, [255].Status := 2, [256].Status := 2, [257].Status := 2, [258].Status := 2, [259].Status := 2, [260].Status := 2, [261].Status := 2, [262].Status := 2, [263].Status := 2, [264].Status := 2, [265].Status := 2, [266].Status := 2, [267].Status := 2, [268].Status := 2, [269].Status := 2, [270].Status := 2, [271].Status := 2, [272].Status := 2, [273].Status := 2, [274].Status := 2, [275].Status := 2, [276].Status := 2, [277].Status := 2, [278].Status := 2, [279].Status := 2, [280].Status := 2, [281].Status := 2, [282].Status := 2, [283].Status := 2, [284].Status := 2, [285].Status := 2, [286].Status := 2, [287].Status := 2, [288].Status := 2, [289].Status := 2, [290].Status := 2, [291].Status := 2, [292].Status := 2, [293].Status := 2, [294].Status := 2, [295].Status := 2, [296].Status := 2, [297].Status := 2, [298].Status := 2, [299].Status := 2,
        [300].Status := 2, [301].Status := 2, [302].Status := 2, [303].Status := 2, [304].Status := 2, [305].Status := 2, [306].Status := 2, [307].Status := 2, [308].Status := 2, [309].Status := 2, [310].Status := 2, [311].Status := 2, [312].Status := 2, [313].Status := 2, [314].Status := 2, [315].Status := 2, [316].Status := 2, [317].Status := 2, [318].Status := 2, [319].Status := 2, [320].Status := 2, [321].Status := 2, [322].Status := 2, [323].Status := 2, [324].Status := 2, [325].Status := 2, [326].Status := 2, [327].Status := 2, [328].Status := 2, [329].Status := 2, [330].Status := 2, [331].Status := 2, [332].Status := 2, [333].Status := 2, [334].Status := 2, [335].Status := 2, [336].Status := 2, [337].Status := 2, [338].Status := 2, [339].Status := 2, [340].Status := 2, [341].Status := 2, [342].Status := 2, [343].Status := 2, [344].Status := 2, [345].Status := 2, [346].Status := 2, [347].Status := 2, [348].Status := 2, [349].Status := 2, [350].Status := 2, [351].Status := 2, [352].Status := 2, [353].Status := 2, [354].Status := 2, [355].Status := 2, [356].Status := 2, [357].Status := 2, [358].Status := 2, [359].Status := 2,
        [360].Status := 2, [361].Status := 2, [362].Status := 2, [363].Status := 2, [364].Status := 2, [365].Status := 2, [366].Status := 2, [367].Status := 2, [368].Status := 2, [369].Status := 2, [370].Status := 2, [371].Status := 2, [372].Status := 2, [373].Status := 2, [374].Status := 2, [375].Status := 2, [376].Status := 2, [377].Status := 2, [378].Status := 2, [379].Status := 2, [380].Status := 2, [381].Status := 2, [382].Status := 2, [383].Status := 2, [384].Status := 2, [385].Status := 2, [386].Status := 2, [387].Status := 2, [388].Status := 2, [389].Status := 2, [390].Status := 2, [391].Status := 2, [392].Status := 2, [393].Status := 2, [394].Status := 2, [395].Status := 2, [396].Status := 2, [397].Status := 2, [398].Status := 2, [399].Status := 2, [400].Status := 2, [401].Status := 2, [402].Status := 2, [403].Status := 2, [404].Status := 2, [405].Status := 2, [406].Status := 2, [407].Status := 2, [408].Status := 2, [409].Status := 2, [410].Status := 2, [411].Status := 2, [412].Status := 2, [413].Status := 2, [414].Status := 2, [415].Status := 2, [416].Status := 2, [417].Status := 2, [418].Status := 2, [419].Status := 2,
        [420].Status := 2, [421].Status := 2, [422].Status := 2, [423].Status := 2, [424].Status := 2, [425].Status := 2, [426].Status := 2, [427].Status := 2, [428].Status := 2, [429].Status := 2, [430].Status := 2, [431].Status := 2, [432].Status := 2, [433].Status := 2, [434].Status := 2, [435].Status := 2, [436].Status := 2, [437].Status := 2, [438].Status := 2, [439].Status := 2, [440].Status := 2, [441].Status := 2, [442].Status := 2, [443].Status := 2, [444].Status := 2, [445].Status := 2, [446].Status := 2, [447].Status := 2, [448].Status := 2, [449].Status := 2, [450].Status := 2, [451].Status := 2, [452].Status := 2, [453].Status := 2, [454].Status := 2, [455].Status := 2, [456].Status := 2, [457].Status := 2, [458].Status := 2, [459].Status := 2, [460].Status := 2, [461].Status := 2, [462].Status := 2, [463].Status := 2, [464].Status := 2, [465].Status := 2, [466].Status := 2, [467].Status := 2, [468].Status := 2, [469].Status := 2, [470].Status := 2, [471].Status := 2, [472].Status := 2, [473].Status := 2, [474].Status := 2, [475].Status := 2, [476].Status := 2, [477].Status := 2, [478].Status := 2, [479].Status := 2,
        [480].Status := 2, [481].Status := 2, [482].Status := 2, [483].Status := 2, [484].Status := 2, [485].Status := 2, [486].Status := 2, [487].Status := 2, [488].Status := 2, [489].Status := 2, [490].Status := 2, [491].Status := 2, [492].Status := 2, [493].Status := 2, [494].Status := 2, [495].Status := 2, [496].Status := 2, [497].Status := 2, [498].Status := 2, [499].Status := 2, [500].Status := 2, [501].Status := 2, [502].Status := 2, [503].Status := 2, [504].Status := 2, [505].Status := 2, [506].Status := 2, [507].Status := 2, [508].Status := 2, [509].Status := 2, [510].Status := 2, [511].Status := 2, [512].Status := 2, [513].Status := 2, [514].Status := 2, [515].Status := 2, [516].Status := 2, [517].Status := 2, [518].Status := 2, [519].Status := 2, [520].Status := 2, [521].Status := 2, [522].Status := 2, [523].Status := 2, [524].Status := 2, [525].Status := 2, [526].Status := 2, [527].Status := 2, [528].Status := 2, [529].Status := 2, [530].Status := 2, [531].Status := 2, [532].Status := 2, [533].Status := 2, [534].Status := 2, [535].Status := 2, [536].Status := 2, [537].Status := 2, [538].Status := 2, [539].Status := 2,
        [540].Status := 2, [541].Status := 2, [542].Status := 2, [543].Status := 2, [544].Status := 2, [545].Status := 2, [546].Status := 2, [547].Status := 2, [548].Status := 2, [549].Status := 2, [550].Status := 2, [551].Status := 2, [552].Status := 2, [553].Status := 2, [554].Status := 2, [555].Status := 2, [556].Status := 2, [557].Status := 2, [558].Status := 2, [559].Status := 2, [560].Status := 2, [561].Status := 2, [562].Status := 2, [563].Status := 2, [564].Status := 2, [565].Status := 2, [566].Status := 2, [567].Status := 2, [568].Status := 2, [569].Status := 2, [570].Status := 2, [571].Status := 2, [572].Status := 2, [573].Status := 2, [574].Status := 2, [575].Status := 2, [576].Status := 2, [577].Status := 2, [578].Status := 2, [579].Status := 2, [580].Status := 2, [581].Status := 2, [582].Status := 2, [583].Status := 2, [584].Status := 2, [585].Status := 2, [586].Status := 2, [587].Status := 2, [588].Status := 2, [589].Status := 2, [590].Status := 2, [591].Status := 2, [592].Status := 2, [593].Status := 2, [594].Status := 2, [595].Status := 2, [596].Status := 2, [597].Status := 2, [598].Status := 2, [599].Status := 2,
